                    IF (((( NOT ChargeMode) OR DriveMode) OR SDError_BB) OR (BoxAvailable = 0.0)) AND ( NOT HV_REL_ON_BB) THEN 
                        (* Transition: '<S53>:21' *)
                        (* Exit Internal 'CHARGE': '<S53>:46' *)
                        is_CHARGE := ChiefMaster_IN_NO_ACTIVE_CHILD_jz;
                        is_c66_ChiefMaster := ChiefMaster_IN_Default_d;
                        (* Entry 'Default': '<S53>:9' *)
                        (* '<S53>:9:2' REQ_IMD_ON = false; *)
                        REQ_IMD_ON := FALSE;
                        (* '<S53>:9:3' IMD_State = uint8(0); *)
                        IMD_State := 0;
                    ELSE 

                        CASE is_CHARGE OF
                            ChiefMaster_IN_CHARGE_c: 
                                (* During 'CHARGE': '<S53>:13' *)
                                (* '<S53>:32:1' sf_internal_predicateOutput = InsulationReadyOK == true &&... *)
                                (* '<S53>:32:2' MinVtgBB == BattNo &&... *)
                                (* '<S53>:32:3' HV_ON_BB == false; *)

                                IF (InsulationReadyOK AND (MinVtgBB = BattNo)) AND ( NOT HV_ON_BB) THEN 
                                    (* Transition: '<S53>:32' *)
                                    is_CHARGE := ChiefMaster_IN_IMD_ON_b;
                                    (* Entry 'IMD_ON': '<S53>:31' *)
                                    (* '<S53>:31:2' REQ_IMD_ON = true; *)
                                    REQ_IMD_ON := TRUE;
                                    (* '<S53>:31:3' IMD_State = uint8(5); *)
                                    IMD_State := 5;
                                ELSE 
                                    (* '<S53>:34:1' sf_internal_predicateOutput = (InsulationReadyOK == true && MinVtgBB ~=  BattNo) ||... *)
                                    (* '<S53>:34:2'  HV_ON_BB == true; *)

                                    IF (InsulationReadyOK AND (MinVtgBB <> BattNo)) OR HV_ON_BB THEN 
                                        (* Transition: '<S53>:34' *)
                                        is_CHARGE := ChiefMaster_IN_IMD_OFF_m;
                                        (* Entry 'IMD_OFF': '<S53>:33' *)
                                        (* '<S53>:33:2' REQ_IMD_ON = false; *)
                                        REQ_IMD_ON := FALSE;
                                        (* '<S53>:33:3' IMD_State = uint8(6); *)
                                        IMD_State := 6;
                                    ELSE 
                                        (* '<S53>:13:2' REQ_IMD_ON = true; *)
                                        REQ_IMD_ON := TRUE;
                                        (* '<S53>:13:3' IMD_State = uint8(4); *)
                                        IMD_State := 4;
                                    END_IF;

                                END_IF;

                            ChiefMaster_IN_IMD_OFF_m: 
                                (* During 'IMD_OFF': '<S53>:33' *)
                                (* '<S53>:75:1' sf_internal_predicateOutput = MinVtgBB == BattNo &&... *)
                                (* '<S53>:75:2' IMD_Active_BB1 == false &&... *)
                                (* '<S53>:75:3' IMD_Active_BB2 == false &&... *)
                                (* '<S53>:75:4' IMD_Active_BB3 == false &&... *)
                                (* '<S53>:75:5' IsolationMeasurementRequest == true; *)

                                IF ((((MinVtgBB = BattNo) AND ( NOT IMD_Active_BB1)) AND ( NOT IMD_Active_BB2)) AND ( NOT IMD_Active_BB3)) AND IsolationMeasurementRequest THEN 
                                    (* Transition: '<S53>:75' *)
                                    is_CHARGE := ChiefMaster_IN_IMD_ON_b;
                                    (* Entry 'IMD_ON': '<S53>:31' *)
                                    (* '<S53>:31:2' REQ_IMD_ON = true; *)
                                    REQ_IMD_ON := TRUE;
                                    (* '<S53>:31:3' IMD_State = uint8(5); *)
                                    IMD_State := 5;
                                ELSE 
                                    (* '<S53>:33:2' REQ_IMD_ON = false; *)
                                    REQ_IMD_ON := FALSE;
                                    (* '<S53>:33:3' IMD_State = uint8(6); *)
                                    IMD_State := 6;
                                END_IF;

                            ELSE
                                (* During 'IMD_ON': '<S53>:31' *)
                                (* '<S53>:87:1' sf_internal_predicateOutput = HV_ON_BB == true &&... *)
                                (* '<S53>:87:2' IsolationMeasurementRequest == false; *)

                                IF HV_ON_BB AND ( NOT IsolationMeasurementRequest) THEN 
                                    (* Transition: '<S53>:87' *)
                                    is_CHARGE := ChiefMaster_IN_IMD_OFF_m;
                                    (* Entry 'IMD_OFF': '<S53>:33' *)
                                    (* '<S53>:33:2' REQ_IMD_ON = false; *)
                                    REQ_IMD_ON := FALSE;
                                    (* '<S53>:33:3' IMD_State = uint8(6); *)
                                    IMD_State := 6;
                                ELSE 
                                    (* '<S53>:31:2' REQ_IMD_ON = true; *)
                                    REQ_IMD_ON := TRUE;
                                    (* '<S53>:31:3' IMD_State = uint8(5); *)
                                    IMD_State := 5;
                                END_IF;

                        END_CASE;

                    END_IF;

                ChiefMaster_IN_DRIVE_k: 
                    (* During 'DRIVE': '<S53>:62' *)
                    (* '<S53>:27:1' sf_internal_predicateOutput = ((DriveMode == false || ChargeMode == true ||... *)
                    (* '<S53>:27:2' SDError_BB == true || BoxAvailable==false) &&... *)
                    (* '<S53>:27:3' HV_REL_ON_BB == false); *)

                    IF (((( NOT DriveMode) OR ChargeMode) OR SDError_BB) OR (BoxAvailable = 0.0)) AND ( NOT HV_REL_ON_BB) THEN 
                        (* Transition: '<S53>:27' *)
                        (* Exit Internal 'DRIVE': '<S53>:62' *)
                        is_DRIVE := ChiefMaster_IN_NO_ACTIVE_CHILD_jz;
                        is_c66_ChiefMaster := ChiefMaster_IN_Default_d;
                        (* Entry 'Default': '<S53>:9' *)
                        (* '<S53>:9:2' REQ_IMD_ON = false; *)
                        REQ_IMD_ON := FALSE;
                        (* '<S53>:9:3' IMD_State = uint8(0); *)
                        IMD_State := 0;
                    ELSE 

                        CASE is_DRIVE OF
                            ChiefMaster_IN_DRIVE_ke: 
                                (* During 'DRIVE': '<S53>:63' *)
                                (* '<S53>:67:1' sf_internal_predicateOutput = InsulationReadyOK == true &&... *)
                                (* '<S53>:67:2' MaxVtgBB == BattNo &&... *)
                                (* '<S53>:67:3' HV_ON_BB == false; *)

                                IF (InsulationReadyOK AND (MaxVtgBB = BattNo)) AND ( NOT HV_ON_BB) THEN 
                                    (* Transition: '<S53>:67' *)
                                    is_DRIVE := ChiefMaster_IN_IMD_ON_b;
                                    (* Entry 'IMD_ON': '<S53>:64' *)
                                    (* '<S53>:64:2' REQ_IMD_ON = true; *)
                                    REQ_IMD_ON := TRUE;
                                    (* '<S53>:64:3' IMD_State = uint8(2); *)
                                    IMD_State := 2;
                                ELSE 
                                    (* '<S53>:68:1' sf_internal_predicateOutput = (InsulationReadyOK == true && MaxVtgBB ~=  BattNo)  ||... *)
                                    (* '<S53>:68:2' HV_ON_BB == true; *)

                                    IF (InsulationReadyOK AND (MaxVtgBB <> BattNo)) OR HV_ON_BB THEN 
                                        (* Transition: '<S53>:68' *)
                                        is_DRIVE := ChiefMaster_IN_IMD_OFF_m;
                                        (* Entry 'IMD_OFF': '<S53>:65' *)
                                        (* '<S53>:65:2' REQ_IMD_ON = false; *)
                                        REQ_IMD_ON := FALSE;
                                        (* '<S53>:65:3' IMD_State = uint8(3); *)
                                        IMD_State := 3;
                                    ELSE 
                                        (* '<S53>:63:2' REQ_IMD_ON = true; *)
                                        REQ_IMD_ON := TRUE;
                                        (* '<S53>:63:3' IMD_State = uint8(1); *)
                                        IMD_State := 1;
                                    END_IF;

                                END_IF;

                            ChiefMaster_IN_IMD_OFF_m: 
                                (* During 'IMD_OFF': '<S53>:65' *)
                                (* '<S53>:77:1' sf_internal_predicateOutput = MaxVtgBB == BattNo &&... *)
                                (* '<S53>:77:2' IMD_Active_BB1 == false &&... *)
                                (* '<S53>:77:3' IMD_Active_BB2 == false &&... *)
                                (* '<S53>:77:4' IMD_Active_BB3 == false &&... *)
                                (* '<S53>:77:5' IsolationMeasurementRequest == true; *)

                                IF ((((MaxVtgBB = BattNo) AND ( NOT IMD_Active_BB1)) AND ( NOT IMD_Active_BB2)) AND ( NOT IMD_Active_BB3)) AND IsolationMeasurementRequest THEN 
                                    (* Transition: '<S53>:77' *)
                                    is_DRIVE := ChiefMaster_IN_IMD_ON_b;
                                    (* Entry 'IMD_ON': '<S53>:64' *)
                                    (* '<S53>:64:2' REQ_IMD_ON = true; *)
                                    REQ_IMD_ON := TRUE;
                                    (* '<S53>:64:3' IMD_State = uint8(2); *)
                                    IMD_State := 2;
                                ELSE 
                                    (* '<S53>:65:2' REQ_IMD_ON = false; *)
                                    REQ_IMD_ON := FALSE;
                                    (* '<S53>:65:3' IMD_State = uint8(3); *)
                                    IMD_State := 3;
                                END_IF;

                            ELSE
                                (* During 'IMD_ON': '<S53>:64' *)
                                (* '<S53>:88:1' sf_internal_predicateOutput = HV_ON_BB == true &&... *)
                                (* '<S53>:88:2' IsolationMeasurementRequest == false; *)

                                IF HV_ON_BB AND ( NOT IsolationMeasurementRequest) THEN 
                                    (* Transition: '<S53>:88' *)
                                    is_DRIVE := ChiefMaster_IN_IMD_OFF_m;
                                    (* Entry 'IMD_OFF': '<S53>:65' *)
                                    (* '<S53>:65:2' REQ_IMD_ON = false; *)
                                    REQ_IMD_ON := FALSE;
                                    (* '<S53>:65:3' IMD_State = uint8(3); *)
                                    IMD_State := 3;
                                ELSE 
                                    (* '<S53>:64:2' REQ_IMD_ON = true; *)
                                    REQ_IMD_ON := TRUE;
                                    (* '<S53>:64:3' IMD_State = uint8(2); *)
                                    IMD_State := 2;
                                END_IF;

                        END_CASE;

                    END_IF;

                ELSE
                    (* During 'Default': '<S53>:9' *)
                    (* '<S53>:14:1' sf_internal_predicateOutput = ChargeMode == true && DriveMode == false &&... *)
                    (* '<S53>:14:2'  SDError_BB == false && BoxAvailable==true; *)
                    tmp :=  NOT SDError_BB;

                    IF ((ChargeMode AND ( NOT DriveMode)) AND tmp) AND (BoxAvailable = 1.0) THEN 
                        (* Transition: '<S53>:14' *)
                        is_c66_ChiefMaster := ChiefMaster_IN_CHARGE_c;
                        (* Entry Internal 'CHARGE': '<S53>:46' *)
                        (* Transition: '<S53>:47' *)
                        is_CHARGE := ChiefMaster_IN_CHARGE_c;
                        (* Entry 'CHARGE': '<S53>:13' *)
                        (* '<S53>:13:2' REQ_IMD_ON = true; *)
                        REQ_IMD_ON := TRUE;
                        (* '<S53>:13:3' IMD_State = uint8(4); *)
                        IMD_State := 4;
                    ELSE 
                        (* '<S53>:18:1' sf_internal_predicateOutput = DriveMode == true && ChargeMode == false &&... *)
                        (* '<S53>:18:2'  SDError_BB == false && BoxAvailable==true; *)

                        IF ((DriveMode AND ( NOT ChargeMode)) AND tmp) AND (BoxAvailable = 1.0) THEN 
                            (* Transition: '<S53>:18' *)
                            is_c66_ChiefMaster := ChiefMaster_IN_DRIVE_k;
                            (* Entry Internal 'DRIVE': '<S53>:62' *)
                            (* Transition: '<S53>:66' *)
                            is_DRIVE := ChiefMaster_IN_DRIVE_ke;
                            (* Entry 'DRIVE': '<S53>:63' *)
                            (* '<S53>:63:2' REQ_IMD_ON = true; *)
                            REQ_IMD_ON := TRUE;
                            (* '<S53>:63:3' IMD_State = uint8(1); *)
                            IMD_State := 1;
                        ELSE 
                            (* '<S53>:9:2' REQ_IMD_ON = false; *)
                            REQ_IMD_ON := FALSE;
                            (* '<S53>:9:3' IMD_State = uint8(0); *)
                            IMD_State := 0;
                        END_IF;

                    END_IF;

            END_CASE;

        END_IF;

        (* End of Chart: '<S48>/Chart_REQ_IMD_ON_BB2' *)
END_CASE;

END_FUNCTION_BLOCK

// Device/Application/Chart_REQ_IMD_ON_BB3
FUNCTION_BLOCK Chart_REQ_IMD_ON_BB3
VAR_INPUT
	ssMethodType: SINT;
	ChargeMode: BOOL;
	DriveMode: BOOL;
	InsulationReadyOK: BOOL;
	MaxVtgBB: REAL;
	MinVtgBB: REAL;
	SDError_BB: BOOL;
	BattNo: REAL;
	HV_ON_BB: BOOL;
	IMD_Active_BB2: BOOL;
	IMD_Active_BB3: BOOL;
	IMD_Active_BB1: BOOL;
	HV_REL_ON_BB: BOOL;
	BoxAvailable: LREAL;
	IsolationMeasurementRequest: BOOL;
END_VAR
VAR_OUTPUT
	REQ_IMD_ON: BOOL;
	IMD_State: USINT;
END_VAR
VAR
	is_c67_ChiefMaster: USINT;
	is_active_c67_ChiefMaster: USINT;
	is_DRIVE: USINT;
	is_CHARGE: USINT;
	tmp: BOOL;
END_VAR



CASE ssMethodType OF
    SS_INITIALIZE: 
        is_CHARGE := ChiefMaster_IN_NO_ACTIVE_CHILD_g;
        is_DRIVE := ChiefMaster_IN_NO_ACTIVE_CHILD_g;
        is_active_c67_ChiefMaster := 0;
        is_c67_ChiefMaster := ChiefMaster_IN_NO_ACTIVE_CHILD_g;
        REQ_IMD_ON := FALSE;
        IMD_State := 0;
    SS_OUTPUT: 
        (* Chart: '<S48>/Chart_REQ_IMD_ON_BB3' *)
        (* Gateway: ChiefMaster/Flow Logic/IMD Control/InsulationMonitoringReq/Chart_REQ_IMD_ON_BB3 *)
        (* During: ChiefMaster/Flow Logic/IMD Control/InsulationMonitoringReq/Chart_REQ_IMD_ON_BB3 *)

        IF is_active_c67_ChiefMaster = 0 THEN 
            (* Entry: ChiefMaster/Flow Logic/IMD Control/InsulationMonitoringReq/Chart_REQ_IMD_ON_BB3 *)
            is_active_c67_ChiefMaster := 1;
            (* Entry Internal: ChiefMaster/Flow Logic/IMD Control/InsulationMonitoringReq/Chart_REQ_IMD_ON_BB3 *)
            (* Transition: '<S54>:10' *)
            is_c67_ChiefMaster := ChiefMaster_IN_Default_j;
            (* Entry 'Default': '<S54>:9' *)
            (* '<S54>:9:2' REQ_IMD_ON = false; *)
            REQ_IMD_ON := FALSE;
            (* '<S54>:9:3' IMD_State = uint8(0); *)
            IMD_State := 0;
        ELSE 

            CASE is_c67_ChiefMaster OF
                ChiefMaster_IN_CHARGE_a: 
                    (* During 'CHARGE': '<S54>:46' *)
                    (* '<S54>:21:1' sf_internal_predicateOutput = ((ChargeMode == false || DriveMode == true ||... *)
                    (* '<S54>:21:2'  SDError_BB == true || BoxAvailable==false) &&... *)
                    (* '<S54>:21:3' HV_REL_ON_BB == false); *)

                    IF (((( NOT ChargeMode) OR DriveMode) OR SDError_BB) OR (BoxAvailable = 0.0)) AND ( NOT HV_REL_ON_BB) THEN 
                        (* Transition: '<S54>:21' *)
                        (* Exit Internal 'CHARGE': '<S54>:46' *)
                        is_CHARGE := ChiefMaster_IN_NO_ACTIVE_CHILD_g;
                        is_c67_ChiefMaster := ChiefMaster_IN_Default_j;
                        (* Entry 'Default': '<S54>:9' *)
                        (* '<S54>:9:2' REQ_IMD_ON = false; *)
                        REQ_IMD_ON := FALSE;
                        (* '<S54>:9:3' IMD_State = uint8(0); *)
                        IMD_State := 0;
                    ELSE 

                        CASE is_CHARGE OF
                            ChiefMaster_IN_CHARGE_a: 
                                (* During 'CHARGE': '<S54>:13' *)
                                (* '<S54>:32:1' sf_internal_predicateOutput = InsulationReadyOK == true &&... *)
                                (* '<S54>:32:2' MinVtgBB == BattNo &&... *)
                                (* '<S54>:32:3' HV_ON_BB == false; *)

                                IF (InsulationReadyOK AND (MinVtgBB = BattNo)) AND ( NOT HV_ON_BB) THEN 
                                    (* Transition: '<S54>:32' *)
                                    is_CHARGE := ChiefMaster_IN_IMD_ON_k;
                                    (* Entry 'IMD_ON': '<S54>:31' *)
                                    (* '<S54>:31:2' REQ_IMD_ON = true; *)
                                    REQ_IMD_ON := TRUE;
                                    (* '<S54>:31:3' IMD_State = uint8(5); *)
                                    IMD_State := 5;
                                ELSE 
                                    (* '<S54>:34:1' sf_internal_predicateOutput = (InsulationReadyOK == true && MinVtgBB ~=  BattNo) ||... *)
                                    (* '<S54>:34:2'  HV_ON_BB == true; *)

                                    IF (InsulationReadyOK AND (MinVtgBB <> BattNo)) OR HV_ON_BB THEN 
                                        (* Transition: '<S54>:34' *)
                                        is_CHARGE := ChiefMaster_IN_IMD_OFF_a;
                                        (* Entry 'IMD_OFF': '<S54>:33' *)
                                        (* '<S54>:33:2' REQ_IMD_ON = false; *)
                                        REQ_IMD_ON := FALSE;
                                        (* '<S54>:33:3' IMD_State = uint8(6); *)
                                        IMD_State := 6;
                                    ELSE 
                                        (* '<S54>:13:2' REQ_IMD_ON = true; *)
                                        REQ_IMD_ON := TRUE;
                                        (* '<S54>:13:3' IMD_State = uint8(4); *)
                                        IMD_State := 4;
                                    END_IF;

                                END_IF;

                            ChiefMaster_IN_IMD_OFF_a: 
                                (* During 'IMD_OFF': '<S54>:33' *)
                                (* '<S54>:75:1' sf_internal_predicateOutput = MinVtgBB == BattNo &&... *)
                                (* '<S54>:75:2' IMD_Active_BB1 == false &&... *)
                                (* '<S54>:75:3' IMD_Active_BB2 == false &&... *)
                                (* '<S54>:75:4' IMD_Active_BB3 == false &&... *)
                                (* '<S54>:75:5' IsolationMeasurementRequest == true; *)

                                IF ((((MinVtgBB = BattNo) AND ( NOT IMD_Active_BB1)) AND ( NOT IMD_Active_BB2)) AND ( NOT IMD_Active_BB3)) AND IsolationMeasurementRequest THEN 
                                    (* Transition: '<S54>:75' *)
                                    is_CHARGE := ChiefMaster_IN_IMD_ON_k;
                                    (* Entry 'IMD_ON': '<S54>:31' *)
                                    (* '<S54>:31:2' REQ_IMD_ON = true; *)
                                    REQ_IMD_ON := TRUE;
                                    (* '<S54>:31:3' IMD_State = uint8(5); *)
                                    IMD_State := 5;
                                ELSE 
                                    (* '<S54>:33:2' REQ_IMD_ON = false; *)
                                    REQ_IMD_ON := FALSE;
                                    (* '<S54>:33:3' IMD_State = uint8(6); *)
                                    IMD_State := 6;
                                END_IF;

                            ELSE
                                (* During 'IMD_ON': '<S54>:31' *)
                                (* '<S54>:87:1' sf_internal_predicateOutput = HV_ON_BB == true &&... *)
                                (* '<S54>:87:2' IsolationMeasurementRequest == false; *)

                                IF HV_ON_BB AND ( NOT IsolationMeasurementRequest) THEN 
                                    (* Transition: '<S54>:87' *)
                                    is_CHARGE := ChiefMaster_IN_IMD_OFF_a;
                                    (* Entry 'IMD_OFF': '<S54>:33' *)
                                    (* '<S54>:33:2' REQ_IMD_ON = false; *)
                                    REQ_IMD_ON := FALSE;
                                    (* '<S54>:33:3' IMD_State = uint8(6); *)
                                    IMD_State := 6;
                                ELSE 
                                    (* '<S54>:31:2' REQ_IMD_ON = true; *)
                                    REQ_IMD_ON := TRUE;
                                    (* '<S54>:31:3' IMD_State = uint8(5); *)
                                    IMD_State := 5;
                                END_IF;

                        END_CASE;

                    END_IF;

                ChiefMaster_IN_DRIVE_e: 
                    (* During 'DRIVE': '<S54>:62' *)
                    (* '<S54>:27:1' sf_internal_predicateOutput = ((DriveMode == false || ChargeMode == true ||... *)
                    (* '<S54>:27:2' SDError_BB == true || BoxAvailable==false) &&... *)
                    (* '<S54>:27:3' HV_REL_ON_BB == false); *)

                    IF (((( NOT DriveMode) OR ChargeMode) OR SDError_BB) OR (BoxAvailable = 0.0)) AND ( NOT HV_REL_ON_BB) THEN 
                        (* Transition: '<S54>:27' *)
                        (* Exit Internal 'DRIVE': '<S54>:62' *)
                        is_DRIVE := ChiefMaster_IN_NO_ACTIVE_CHILD_g;
                        is_c67_ChiefMaster := ChiefMaster_IN_Default_j;
                        (* Entry 'Default': '<S54>:9' *)
                        (* '<S54>:9:2' REQ_IMD_ON = false; *)
                        REQ_IMD_ON := FALSE;
                        (* '<S54>:9:3' IMD_State = uint8(0); *)
                        IMD_State := 0;
                    ELSE 

                        CASE is_DRIVE OF
                            ChiefMaster_IN_DRIVE_e3: 
                                (* During 'DRIVE': '<S54>:63' *)
                                (* '<S54>:67:1' sf_internal_predicateOutput = InsulationReadyOK == true &&... *)
                                (* '<S54>:67:2' MaxVtgBB == BattNo &&... *)
                                (* '<S54>:67:3' HV_ON_BB == false; *)

                                IF (InsulationReadyOK AND (MaxVtgBB = BattNo)) AND ( NOT HV_ON_BB) THEN 
                                    (* Transition: '<S54>:67' *)
                                    is_DRIVE := ChiefMaster_IN_IMD_ON_k;
                                    (* Entry 'IMD_ON': '<S54>:64' *)
                                    (* '<S54>:64:2' REQ_IMD_ON = true; *)
                                    REQ_IMD_ON := TRUE;
                                    (* '<S54>:64:3' IMD_State = uint8(2); *)
                                    IMD_State := 2;
                                ELSE 
                                    (* '<S54>:68:1' sf_internal_predicateOutput = (InsulationReadyOK == true && MaxVtgBB ~=  BattNo)  ||... *)
                                    (* '<S54>:68:2' HV_ON_BB == true; *)

                                    IF (InsulationReadyOK AND (MaxVtgBB <> BattNo)) OR HV_ON_BB THEN 
                                        (* Transition: '<S54>:68' *)
                                        is_DRIVE := ChiefMaster_IN_IMD_OFF_a;
                                        (* Entry 'IMD_OFF': '<S54>:65' *)
                                        (* '<S54>:65:2' REQ_IMD_ON = false; *)
                                        REQ_IMD_ON := FALSE;
                                        (* '<S54>:65:3' IMD_State = uint8(3); *)
                                        IMD_State := 3;
                                    ELSE 
                                        (* '<S54>:63:2' REQ_IMD_ON = true; *)
                                        REQ_IMD_ON := TRUE;
                                        (* '<S54>:63:3' IMD_State = uint8(1); *)
                                        IMD_State := 1;
                                    END_IF;

                                END_IF;

                            ChiefMaster_IN_IMD_OFF_a: 
                                (* During 'IMD_OFF': '<S54>:65' *)
                                (* '<S54>:77:1' sf_internal_predicateOutput = MaxVtgBB == BattNo &&... *)
                                (* '<S54>:77:2' IMD_Active_BB1 == false &&... *)
                                (* '<S54>:77:3' IMD_Active_BB2 == false &&... *)
                                (* '<S54>:77:4' IMD_Active_BB3 == false &&... *)
                                (* '<S54>:77:5' IsolationMeasurementRequest == true; *)

                                IF ((((MaxVtgBB = BattNo) AND ( NOT IMD_Active_BB1)) AND ( NOT IMD_Active_BB2)) AND ( NOT IMD_Active_BB3)) AND IsolationMeasurementRequest THEN 
                                    (* Transition: '<S54>:77' *)
                                    is_DRIVE := ChiefMaster_IN_IMD_ON_k;
                                    (* Entry 'IMD_ON': '<S54>:64' *)
                                    (* '<S54>:64:2' REQ_IMD_ON = true; *)
                                    REQ_IMD_ON := TRUE;
                                    (* '<S54>:64:3' IMD_State = uint8(2); *)
                                    IMD_State := 2;
                                ELSE 
                                    (* '<S54>:65:2' REQ_IMD_ON = false; *)
                                    REQ_IMD_ON := FALSE;
                                    (* '<S54>:65:3' IMD_State = uint8(3); *)
                                    IMD_State := 3;
                                END_IF;

                            ELSE
                                (* During 'IMD_ON': '<S54>:64' *)
                                (* '<S54>:88:1' sf_internal_predicateOutput = HV_ON_BB == true &&... *)
                                (* '<S54>:88:2' IsolationMeasurementRequest == false; *)

                                IF HV_ON_BB AND ( NOT IsolationMeasurementRequest) THEN 
                                    (* Transition: '<S54>:88' *)
                                    is_DRIVE := ChiefMaster_IN_IMD_OFF_a;
                                    (* Entry 'IMD_OFF': '<S54>:65' *)
                                    (* '<S54>:65:2' REQ_IMD_ON = false; *)
                                    REQ_IMD_ON := FALSE;
                                    (* '<S54>:65:3' IMD_State = uint8(3); *)
                                    IMD_State := 3;
                                ELSE 
                                    (* '<S54>:64:2' REQ_IMD_ON = true; *)
                                    REQ_IMD_ON := TRUE;
                                    (* '<S54>:64:3' IMD_State = uint8(2); *)
                                    IMD_State := 2;
                                END_IF;

                        END_CASE;

                    END_IF;

                ELSE
                    (* During 'Default': '<S54>:9' *)
                    (* '<S54>:14:1' sf_internal_predicateOutput = ChargeMode == true && DriveMode == false &&... *)
                    (* '<S54>:14:2'  SDError_BB == false && BoxAvailable==true; *)
                    tmp :=  NOT SDError_BB;

                    IF ((ChargeMode AND ( NOT DriveMode)) AND tmp) AND (BoxAvailable = 1.0) THEN 
                        (* Transition: '<S54>:14' *)
                        is_c67_ChiefMaster := ChiefMaster_IN_CHARGE_a;
                        (* Entry Internal 'CHARGE': '<S54>:46' *)
                        (* Transition: '<S54>:47' *)
                        is_CHARGE := ChiefMaster_IN_CHARGE_a;
                        (* Entry 'CHARGE': '<S54>:13' *)
                        (* '<S54>:13:2' REQ_IMD_ON = true; *)
                        REQ_IMD_ON := TRUE;
                        (* '<S54>:13:3' IMD_State = uint8(4); *)
                        IMD_State := 4;
                    ELSE 
                        (* '<S54>:18:1' sf_internal_predicateOutput = DriveMode == true && ChargeMode == false &&... *)
                        (* '<S54>:18:2'  SDError_BB == false && BoxAvailable==true; *)

                        IF ((DriveMode AND ( NOT ChargeMode)) AND tmp) AND (BoxAvailable = 1.0) THEN 
                            (* Transition: '<S54>:18' *)
                            is_c67_ChiefMaster := ChiefMaster_IN_DRIVE_e;
                            (* Entry Internal 'DRIVE': '<S54>:62' *)
                            (* Transition: '<S54>:66' *)
                            is_DRIVE := ChiefMaster_IN_DRIVE_e3;
                            (* Entry 'DRIVE': '<S54>:63' *)
                            (* '<S54>:63:2' REQ_IMD_ON = true; *)
                            REQ_IMD_ON := TRUE;
                            (* '<S54>:63:3' IMD_State = uint8(1); *)
                            IMD_State := 1;
                        ELSE 
                            (* '<S54>:9:2' REQ_IMD_ON = false; *)
                            REQ_IMD_ON := FALSE;
                            (* '<S54>:9:3' IMD_State = uint8(0); *)
                            IMD_State := 0;
                        END_IF;

                    END_IF;

            END_CASE;

        END_IF;

        (* End of Chart: '<S48>/Chart_REQ_IMD_ON_BB3' *)
END_CASE;

END_FUNCTION_BLOCK

// Device/Application/PLC_CODER_TIMER
FUNCTION_BLOCK PLC_CODER_TIMER
VAR_INPUT
	timerAction: INT;
	maxTime: DINT;
END_VAR
VAR_OUTPUT
	done: BOOL;
END_VAR
VAR
	plcTimer: TON;
	plcTimerExpired: BOOL;
END_VAR


CASE timerAction OF
    1:
        (* RESET *)
        plcTimer(IN:=FALSE, PT:=T#0ms);
        plcTimerExpired := FALSE;
        done := FALSE;
    2:
        (* AFTER *)
        IF (NOT(plcTimerExpired)) THEN
            plcTimer(IN:=TRUE, PT:=DINT_TO_TIME(maxTime));
        END_IF;
        plcTimerExpired := plcTimer.Q;
        done := plcTimerExpired;
    3:
        (* BEFORE *)
        IF (NOT(plcTimerExpired)) THEN
            plcTimer(IN:=TRUE, PT:=DINT_TO_TIME(maxTime));
        END_IF;
        plcTimerExpired := plcTimer.Q;
        done := NOT(plcTimerExpired);
END_CASE;

END_FUNCTION_BLOCK

// Device/Application/PLC_BOOL_TO_LREAL
FUNCTION PLC_BOOL_TO_LREAL : LREAL
VAR_INPUT
	in: BOOL;
END_VAR
VAR
END_VAR



IF in THEN 
    PLC_BOOL_TO_LREAL := 1.0;
ELSE 
    PLC_BOOL_TO_LREAL := 0.0;
END_IF;

END_FUNCTION

// Device/Application/rt_floord
FUNCTION rt_floord : LREAL
VAR_INPUT
	u: LREAL;
END_VAR
VAR
END_VAR


rt_floord := DINT_TO_LREAL(TRUNC(u));

IF u = rt_floord THEN 
    rt_floord := u;
ELSIF u < 0.0 THEN 
    rt_floord := rt_floord - 1.0;
END_IF;

END_FUNCTION

// Device/Application/rt_floorf
FUNCTION rt_floorf : REAL
VAR_INPUT
	u: REAL;
END_VAR
VAR
END_VAR


rt_floorf := DINT_TO_REAL(TRUNC(u));

IF u = rt_floorf THEN 
    rt_floorf := u;
ELSIF u < 0.0 THEN 
    rt_floorf := rt_floorf - 1.0;
END_IF;

END_FUNCTION

// Device/Application/Chart_m
FUNCTION_BLOCK Chart_m
VAR_INPUT
	ssMethodType: SINT;
	In: BOOL;
	KL15_CM_Reset: BOOL;
END_VAR
VAR_OUTPUT
	Out: BOOL;
END_VAR
VAR
	temporalCounter_i1: PLC_CODER_TIMER;
	is_c45_ChiefMaster: USINT;
	is_active_c45_ChiefMaster: USINT;
END_VAR



CASE ssMethodType OF
    SS_INITIALIZE: 
        temporalCounter_i1(timerAction := 1, maxTime := 0);
        is_active_c45_ChiefMaster := 0;
        is_c45_ChiefMaster := ChiefMaster_IN_NO_ACTIVE_CHILD_mp;
        Out := FALSE;
    SS_OUTPUT: 
        (* Chart: '<S56>/Chart' *)
        (* Gateway: ChiefMaster/Flow Logic/KL15/System_KL15/Subsystem/Chart *)
        (* During: ChiefMaster/Flow Logic/KL15/System_KL15/Subsystem/Chart *)

        IF is_active_c45_ChiefMaster = 0 THEN 
            (* Entry: ChiefMaster/Flow Logic/KL15/System_KL15/Subsystem/Chart *)
            is_active_c45_ChiefMaster := 1;
            (* Entry Internal: ChiefMaster/Flow Logic/KL15/System_KL15/Subsystem/Chart *)
            (* Transition: '<S59>:2' *)
            is_c45_ChiefMaster := ChiefMaster_IN_Default_o;
            temporalCounter_i1(timerAction := 1, maxTime := 0);
            (* Entry 'Default': '<S59>:1' *)
            (* '<S59>:1:2' Out = false *)
            Out := FALSE;
        ELSE 

            CASE is_c45_ChiefMaster OF
                ChiefMaster_IN_Default_o: 
                    (* During 'Default': '<S59>:1' *)
                    (* '<S59>:4:1' sf_internal_predicateOutput = KL15_CM_Reset == false &&... *)
                    (* '<S59>:4:2' after(100,msec); *)

                    IF  NOT KL15_CM_Reset THEN 
                        temporalCounter_i1(timerAction := 2, maxTime := 100);

                        IF temporalCounter_i1.done THEN 
                            (* Transition: '<S59>:4' *)
                            is_c45_ChiefMaster := ChiefMaster_IN_hold_g;
                            (* Entry 'hold': '<S59>:7' *)
                            (* '<S59>:7:2' Out = In *)
                            Out := In;
                        ELSE 
                            (* '<S59>:1:2' Out = false *)
                            Out := FALSE;
                        END_IF;

                    ELSE 
                        (* '<S59>:1:2' Out = false *)
                        Out := FALSE;
                    END_IF;

                ELSE
                    (* During 'hold': '<S59>:7' *)
                    (* '<S59>:7:2' Out = In *)
                    Out := In;
            END_CASE;

        END_IF;

        (* End of Chart: '<S56>/Chart' *)
END_CASE;

END_FUNCTION_BLOCK

// Device/Application/ChartBatt1
FUNCTION_BLOCK ChartBatt1
VAR_INPUT
	ssMethodType: SINT;
	BattAvailable_LiBa: BOOL;
	BattAvailable_Actia: BOOL;
END_VAR
VAR_OUTPUT
	BattSelect: LREAL;
END_VAR
VAR
	is_c9_ChiefMaster: USINT;
	is_active_c9_ChiefMaster: USINT;
END_VAR



CASE ssMethodType OF
    SS_INITIALIZE: 
        is_active_c9_ChiefMaster := 0;
        is_c9_ChiefMaster := ChiefMaster_IN_NO_ACTIVE_CHILD_i3;
        BattSelect := 0.0;
    SS_OUTPUT: 
        (* Chart: '<S675>/ChartBatt1' *)
        (* Gateway: ChiefMaster/Input Translation/Battery Selection/ChartBatt1 *)
        (* During: ChiefMaster/Input Translation/Battery Selection/ChartBatt1 *)

        IF is_active_c9_ChiefMaster = 0 THEN 
            (* Entry: ChiefMaster/Input Translation/Battery Selection/ChartBatt1 *)
            is_active_c9_ChiefMaster := 1;
            (* Entry Internal: ChiefMaster/Input Translation/Battery Selection/ChartBatt1 *)
            (* Transition: '<S679>:2' *)
            is_c9_ChiefMaster := ChiefMaster_IN_Default_at;
            (* Entry 'Default': '<S679>:1' *)
            (* '<S679>:1:2' BattSelect=0; *)
            BattSelect := 0.0;
        ELSE 

            CASE is_c9_ChiefMaster OF
                ChiefMaster_IN_Actia: 
                    (* During 'Actia': '<S679>:3' *)
                    (* '<S679>:7:1' sf_internal_predicateOutput = BattAvailable_Actia == false; *)

                    IF  NOT BattAvailable_Actia THEN 
                        (* Transition: '<S679>:7' *)
                        is_c9_ChiefMaster := ChiefMaster_IN_Default_at;
                        (* Entry 'Default': '<S679>:1' *)
                        (* '<S679>:1:2' BattSelect=0; *)
                        BattSelect := 0.0;
                    ELSE 
                        (* '<S679>:3:2' BattSelect=1; *)
                        BattSelect := 1.0;
                    END_IF;

                ChiefMaster_IN_Default_at: 
                    (* During 'Default': '<S679>:1' *)
                    (* '<S679>:6:1' sf_internal_predicateOutput = BattAvailable_Actia == true &&... *)
                    (* '<S679>:6:2' BattAvailable_LiBa == false; *)

                    IF BattAvailable_Actia AND ( NOT BattAvailable_LiBa) THEN 
                        (* Transition: '<S679>:6' *)
                        is_c9_ChiefMaster := ChiefMaster_IN_Actia;
                        (* Entry 'Actia': '<S679>:3' *)
                        (* '<S679>:3:2' BattSelect=1; *)
                        BattSelect := 1.0;
                    ELSE 
                        (* '<S679>:5:1' sf_internal_predicateOutput = BattAvailable_Actia == false &&... *)
                        (* '<S679>:5:2' BattAvailable_LiBa == true; *)

                        IF ( NOT BattAvailable_Actia) AND BattAvailable_LiBa THEN 
                            (* Transition: '<S679>:5' *)
                            is_c9_ChiefMaster := ChiefMaster_IN_LiBa;
                            (* Entry 'LiBa': '<S679>:4' *)
                            (* '<S679>:4:2' BattSelect = 2; *)
                            BattSelect := 2.0;
                        ELSE 
                            (* '<S679>:1:2' BattSelect=0; *)
                            BattSelect := 0.0;
                        END_IF;

                    END_IF;

                ELSE
                    (* During 'LiBa': '<S679>:4' *)
                    (* '<S679>:8:1' sf_internal_predicateOutput = BattAvailable_LiBa == false; *)

                    IF  NOT BattAvailable_LiBa THEN 
                        (* Transition: '<S679>:8' *)
                        is_c9_ChiefMaster := ChiefMaster_IN_Default_at;
                        (* Entry 'Default': '<S679>:1' *)
                        (* '<S679>:1:2' BattSelect=0; *)
                        BattSelect := 0.0;
                    ELSE 
                        (* '<S679>:4:2' BattSelect = 2; *)
                        BattSelect := 2.0;
                    END_IF;

            END_CASE;

        END_IF;

        (* End of Chart: '<S675>/ChartBatt1' *)
END_CASE;

END_FUNCTION_BLOCK

// Device/Application/Chartbatt2
FUNCTION_BLOCK Chartbatt2
VAR_INPUT
	ssMethodType: SINT;
	BattAvailable_LiBa: BOOL;
	BattAvailable_Actia: BOOL;
END_VAR
VAR_OUTPUT
	BattSelect: LREAL;
END_VAR
VAR
	is_c22_ChiefMaster: USINT;
	is_active_c22_ChiefMaster: USINT;
END_VAR



CASE ssMethodType OF
    SS_INITIALIZE: 
        is_active_c22_ChiefMaster := 0;
        is_c22_ChiefMaster := ChiefMaster_IN_NO_ACTIVE_CHILD_gp;
        BattSelect := 0.0;
    SS_OUTPUT: 
        (* Chart: '<S675>/Chartbatt2' *)
        (* Gateway: ChiefMaster/Input Translation/Battery Selection/Chartbatt2 *)
        (* During: ChiefMaster/Input Translation/Battery Selection/Chartbatt2 *)

        IF is_active_c22_ChiefMaster = 0 THEN 
            (* Entry: ChiefMaster/Input Translation/Battery Selection/Chartbatt2 *)
            is_active_c22_ChiefMaster := 1;
            (* Entry Internal: ChiefMaster/Input Translation/Battery Selection/Chartbatt2 *)
            (* Transition: '<S681>:2' *)
            is_c22_ChiefMaster := ChiefMaster_IN_Default_bc;
            (* Entry 'Default': '<S681>:1' *)
            (* '<S681>:1:2' BattSelect=0; *)
            BattSelect := 0.0;
        ELSE 

            CASE is_c22_ChiefMaster OF
                ChiefMaster_IN_Actia_p: 
                    (* During 'Actia': '<S681>:3' *)
                    (* '<S681>:7:1' sf_internal_predicateOutput = BattAvailable_Actia == false; *)

                    IF  NOT BattAvailable_Actia THEN 
                        (* Transition: '<S681>:7' *)
                        is_c22_ChiefMaster := ChiefMaster_IN_Default_bc;
                        (* Entry 'Default': '<S681>:1' *)
                        (* '<S681>:1:2' BattSelect=0; *)
                        BattSelect := 0.0;
                    ELSE 
                        (* '<S681>:3:2' BattSelect=1; *)
                        BattSelect := 1.0;
                    END_IF;

                ChiefMaster_IN_Default_bc: 
                    (* During 'Default': '<S681>:1' *)
                    (* '<S681>:6:1' sf_internal_predicateOutput = BattAvailable_Actia == true &&... *)
                    (* '<S681>:6:2' BattAvailable_LiBa == false; *)

                    IF BattAvailable_Actia AND ( NOT BattAvailable_LiBa) THEN 
                        (* Transition: '<S681>:6' *)
                        is_c22_ChiefMaster := ChiefMaster_IN_Actia_p;
                        (* Entry 'Actia': '<S681>:3' *)
                        (* '<S681>:3:2' BattSelect=1; *)
                        BattSelect := 1.0;
                    ELSE 
                        (* '<S681>:5:1' sf_internal_predicateOutput = BattAvailable_Actia == false &&... *)
                        (* '<S681>:5:2' BattAvailable_LiBa == true; *)

                        IF ( NOT BattAvailable_Actia) AND BattAvailable_LiBa THEN 
                            (* Transition: '<S681>:5' *)
                            is_c22_ChiefMaster := ChiefMaster_IN_LiBa_d;
                            (* Entry 'LiBa': '<S681>:4' *)
                            (* '<S681>:4:2' BattSelect = 2; *)
                            BattSelect := 2.0;
                        ELSE 
                            (* '<S681>:1:2' BattSelect=0; *)
                            BattSelect := 0.0;
                        END_IF;

                    END_IF;

                ELSE
                    (* During 'LiBa': '<S681>:4' *)
                    (* '<S681>:8:1' sf_internal_predicateOutput = BattAvailable_LiBa == false; *)

                    IF  NOT BattAvailable_LiBa THEN 
                        (* Transition: '<S681>:8' *)
                        is_c22_ChiefMaster := ChiefMaster_IN_Default_bc;
                        (* Entry 'Default': '<S681>:1' *)
                        (* '<S681>:1:2' BattSelect=0; *)
                        BattSelect := 0.0;
                    ELSE 
                        (* '<S681>:4:2' BattSelect = 2; *)
                        BattSelect := 2.0;
                    END_IF;

            END_CASE;

        END_IF;

        (* End of Chart: '<S675>/Chartbatt2' *)
END_CASE;

END_FUNCTION_BLOCK

// Device/Application/ChartBatt3
FUNCTION_BLOCK ChartBatt3
VAR_INPUT
	ssMethodType: SINT;
	BattAvailable_LiBa: BOOL;
	BattAvailable_Actia: BOOL;
END_VAR
VAR_OUTPUT
	BattSelect: LREAL;
END_VAR
VAR
	is_c23_ChiefMaster: USINT;
	is_active_c23_ChiefMaster: USINT;
END_VAR



CASE ssMethodType OF
    SS_INITIALIZE: 
        is_active_c23_ChiefMaster := 0;
        is_c23_ChiefMaster := ChiefMaster_IN_NO_ACTIVE_CHILD_d4;
        BattSelect := 0.0;
    SS_OUTPUT: 
        (* Chart: '<S675>/ChartBatt3' *)
        (* Gateway: ChiefMaster/Input Translation/Battery Selection/ChartBatt3 *)
        (* During: ChiefMaster/Input Translation/Battery Selection/ChartBatt3 *)

        IF is_active_c23_ChiefMaster = 0 THEN 
            (* Entry: ChiefMaster/Input Translation/Battery Selection/ChartBatt3 *)
            is_active_c23_ChiefMaster := 1;
            (* Entry Internal: ChiefMaster/Input Translation/Battery Selection/ChartBatt3 *)
            (* Transition: '<S680>:2' *)
            is_c23_ChiefMaster := ChiefMaster_IN_Default_jw;
            (* Entry 'Default': '<S680>:1' *)
            (* '<S680>:1:2' BattSelect=0; *)
            BattSelect := 0.0;
        ELSE 

            CASE is_c23_ChiefMaster OF
                ChiefMaster_IN_Actia_m: 
                    (* During 'Actia': '<S680>:3' *)
                    (* '<S680>:7:1' sf_internal_predicateOutput = BattAvailable_Actia == false; *)

                    IF  NOT BattAvailable_Actia THEN 
                        (* Transition: '<S680>:7' *)
                        is_c23_ChiefMaster := ChiefMaster_IN_Default_jw;
                        (* Entry 'Default': '<S680>:1' *)
                        (* '<S680>:1:2' BattSelect=0; *)
                        BattSelect := 0.0;
                    ELSE 
                        (* '<S680>:3:2' BattSelect=1; *)
                        BattSelect := 1.0;
                    END_IF;

                ChiefMaster_IN_Default_jw: 
                    (* During 'Default': '<S680>:1' *)
                    (* '<S680>:6:1' sf_internal_predicateOutput = BattAvailable_Actia == true &&... *)
                    (* '<S680>:6:2' BattAvailable_LiBa == false; *)

                    IF BattAvailable_Actia AND ( NOT BattAvailable_LiBa) THEN 
                        (* Transition: '<S680>:6' *)
                        is_c23_ChiefMaster := ChiefMaster_IN_Actia_m;
                        (* Entry 'Actia': '<S680>:3' *)
                        (* '<S680>:3:2' BattSelect=1; *)
                        BattSelect := 1.0;
                    ELSE 
                        (* '<S680>:5:1' sf_internal_predicateOutput = BattAvailable_Actia == false &&... *)
                        (* '<S680>:5:2' BattAvailable_LiBa == true; *)

                        IF ( NOT BattAvailable_Actia) AND BattAvailable_LiBa THEN 
                            (* Transition: '<S680>:5' *)
                            is_c23_ChiefMaster := ChiefMaster_IN_LiBa_h;
                            (* Entry 'LiBa': '<S680>:4' *)
                            (* '<S680>:4:2' BattSelect = 2; *)
                            BattSelect := 2.0;
                        ELSE 
                            (* '<S680>:1:2' BattSelect=0; *)
                            BattSelect := 0.0;
                        END_IF;

                    END_IF;

                ELSE
                    (* During 'LiBa': '<S680>:4' *)
                    (* '<S680>:8:1' sf_internal_predicateOutput = BattAvailable_LiBa == false; *)

                    IF  NOT BattAvailable_LiBa THEN 
                        (* Transition: '<S680>:8' *)
                        is_c23_ChiefMaster := ChiefMaster_IN_Default_jw;
                        (* Entry 'Default': '<S680>:1' *)
                        (* '<S680>:1:2' BattSelect=0; *)
                        BattSelect := 0.0;
                    ELSE 
                        (* '<S680>:4:2' BattSelect = 2; *)
                        BattSelect := 2.0;
                    END_IF;

            END_CASE;

        END_IF;

        (* End of Chart: '<S675>/ChartBatt3' *)
END_CASE;

END_FUNCTION_BLOCK

// Device/Application/Lib_InputProcessing_state
FUNCTION_BLOCK Lib_InputProcessing_state
VAR_INPUT
	ssMethodType: SINT;
	Timeout: BOOL;
	Data_In: USINT;
END_VAR
VAR_OUTPUT
	u8Data_Out: USINT;
END_VAR
VAR
	Lib_InputProcessing_state_MODE: BOOL;
END_VAR



CASE ssMethodType OF
    SS_INITIALIZE: 
        (* SystemInitialize for Outport: '<S481>/u8Data_Out' *)
        u8Data_Out := 0;
    SS_OUTPUT: 
        (* Outputs for Enabled SubSystem: '<S428>/Lib_InputProcessing_state' incorporates:
         *  EnablePort: '<S481>/Timeout' *)

        IF Timeout THEN 

            IF  NOT Lib_InputProcessing_state_MODE THEN 
                Lib_InputProcessing_state_MODE := TRUE;
            END_IF;

            (* DataTypeConversion: '<S481>/Data Type Conversion' *)
            u8Data_Out := Data_In;
        ELSIF Lib_InputProcessing_state_MODE THEN 
            (* Disable for Outport: '<S481>/u8Data_Out' *)
            u8Data_Out := 0;
            Lib_InputProcessing_state_MODE := FALSE;
        END_IF;

        (* End of Outputs for SubSystem: '<S428>/Lib_InputProcessing_state' *)
    SS_DISABLE: 
        (* Disable for Outport: '<S481>/u8Data_Out' *)
        u8Data_Out := 0;
        Lib_InputProcessing_state_MODE := FALSE;
END_CASE;

END_FUNCTION_BLOCK

// Device/Application/IMD_OK
FUNCTION_BLOCK IMD_OK
VAR_INPUT
	ssMethodType: SINT;
	IP_boBMS_InsulationReadyOK: BOOL;
	Req_IMD: BOOL;
	IT_u8IMD_DelayTime_s_g: USINT;
END_VAR
VAR_OUTPUT
	IMD_OK_i: BOOL;
END_VAR
VAR
	temporalCounter_i1: PLC_CODER_TIMER;
	is_c63_ChiefMaster: USINT;
	is_active_c63_ChiefMaster: USINT;
	Req_IMD_prev: BOOL;
	Req_IMD_start: BOOL;
END_VAR



CASE ssMethodType OF
    SS_INITIALIZE: 
        temporalCounter_i1(timerAction := 1, maxTime := 0);
        is_active_c63_ChiefMaster := 0;
        is_c63_ChiefMaster := ChiefMaster_IN_NO_ACTIVE_CHILD_gd;
        IMD_OK_i := FALSE;
    SS_OUTPUT: 
        (* Gateway: ChiefMaster/Input Translation/Battery Signals/Subsystem7/Subsystem1/IMD_OK *)
        Req_IMD_prev := Req_IMD_start;
        Req_IMD_start := Req_IMD;
        (* Chart: '<S766>/IMD_OK' *)
        (* During: ChiefMaster/Input Translation/Battery Signals/Subsystem7/Subsystem1/IMD_OK *)

        IF is_active_c63_ChiefMaster = 0 THEN 
            Req_IMD_prev := Req_IMD;
            (* Entry: ChiefMaster/Input Translation/Battery Signals/Subsystem7/Subsystem1/IMD_OK *)
            is_active_c63_ChiefMaster := 1;
            (* Entry Internal: ChiefMaster/Input Translation/Battery Signals/Subsystem7/Subsystem1/IMD_OK *)
            (* Transition: '<S769>:3' *)
            is_c63_ChiefMaster := ChiefMaster_IN_Default_i;
            (* Entry 'Default': '<S769>:2' *)
            (* '<S769>:2:2' IMD_OK=false; *)
            IMD_OK_i := FALSE;
        ELSE 

            CASE is_c63_ChiefMaster OF
                ChiefMaster_IN_Default_i: 
                    (* During 'Default': '<S769>:2' *)
                    (* '<S769>:5:1' sf_internal_predicateOutput = IP_boBMS_InsulationReadyOK == true; *)

                    IF IP_boBMS_InsulationReadyOK THEN 
                        (* Transition: '<S769>:5' *)
                        is_c63_ChiefMaster := ChiefMaster_IN_Hold3;
                        temporalCounter_i1(timerAction := 1, maxTime := 0);
                        (* Entry 'Hold3': '<S769>:23' *)
                        (* '<S769>:23:2' IMD_OK=false; *)
                        IMD_OK_i := FALSE;
                    ELSE 
                        (* '<S769>:2:2' IMD_OK=false; *)
                        IMD_OK_i := FALSE;
                    END_IF;

                ChiefMaster_IN_Hold_m: 
                    (* During 'Hold': '<S769>:4' *)
                    (* '<S769>:19:1' sf_internal_predicateOutput = Req_IMD == false; *)

                    IF  NOT Req_IMD THEN 
                        (* Transition: '<S769>:19' *)
                        is_c63_ChiefMaster := ChiefMaster_IN_Hold2;
                        (* Entry 'Hold2': '<S769>:18' *)
                        (* '<S769>:18:2' IMD_OK=true; *)
                        IMD_OK_i := TRUE;
                    ELSE 
                        (* '<S769>:4:2' IMD_OK=true; *)
                        IMD_OK_i := TRUE;
                    END_IF;

                ChiefMaster_IN_Hold2: 
                    (* During 'Hold2': '<S769>:18' *)
                    (* '<S769>:13:1' sf_internal_predicateOutput = hasChangedFrom(Req_IMD,false); *)

                    IF (Req_IMD_prev <> Req_IMD_start) AND ( NOT Req_IMD_prev) THEN 
                        (* Transition: '<S769>:13' *)
                        (* Transition: '<S769>:26' *)
                        is_c63_ChiefMaster := ChiefMaster_IN_Default_i;
                        (* Entry 'Default': '<S769>:2' *)
                        (* '<S769>:2:2' IMD_OK=false; *)
                        IMD_OK_i := FALSE;
                    ELSE 
                        (* '<S769>:18:2' IMD_OK=true; *)
                        IMD_OK_i := TRUE;
                    END_IF;

                ELSE
                    (* During 'Hold3': '<S769>:23' *)
                    (* '<S769>:24:1' sf_internal_predicateOutput = after(IT_u8IMD_DelayTime_s,sec) &&... *)
                    (* '<S769>:24:2' IP_boBMS_InsulationReadyOK == true; *)
                    temporalCounter_i1(timerAction := 2, maxTime := USINT_TO_DINT(IT_u8IMD_DelayTime_s_g) * 1000);

                    IF temporalCounter_i1.done THEN 

                        IF IP_boBMS_InsulationReadyOK THEN 
                            (* Transition: '<S769>:24' *)
                            is_c63_ChiefMaster := ChiefMaster_IN_Hold_m;
                            (* Entry 'Hold': '<S769>:4' *)
                            (* '<S769>:4:2' IMD_OK=true; *)
                            IMD_OK_i := TRUE;
                        ELSE 
                            (* '<S769>:23:2' IMD_OK=false; *)
                            IMD_OK_i := FALSE;
                        END_IF;

                    ELSE 
                        (* '<S769>:23:2' IMD_OK=false; *)
                        IMD_OK_i := FALSE;
                    END_IF;

            END_CASE;

        END_IF;

        (* End of Chart: '<S766>/IMD_OK' *)
END_CASE;

END_FUNCTION_BLOCK

// Device/Application/REQ_HV_ON_Batt
FUNCTION_BLOCK REQ_HV_ON_Batt
VAR_INPUT
	ssMethodType: SINT;
	IsolationMeasurementRequest: BOOL;
	IP_boChargeStop_Pressed: BOOL;
	SafeToSD_BB1: BOOL;
	SafeToSD_BB2: BOOL;
	SafeToSD_BB3: BOOL;
	KL15_CM_disable: BOOL;
	SDError_BB1: BOOL;
	SDError_BB2: BOOL;
	SDError_BB3: BOOL;
	InsulationReadyOK_B1: BOOL;
	InsulationReadyOK_B2: BOOL;
	InsulationReadyOK_B3: BOOL;
	IMD_Active_BB1: BOOL;
	IMD_Active_BB2: BOOL;
	IMD_Active_BB3: BOOL;
	Software_Reset_KL15_BB3: LREAL;
	Software_Reset_KL15_BB2: LREAL;
	Software_Reset_KL15_BB1: LREAL;
	FL_boSafeToCloseHV_BB1: BOOL;
	FL_boSafeToCloseHV_BB2: BOOL;
	FL_boSafeToCloseHV_BB3: BOOL;
	FL_boST_REQ_HV_Open_BB1: BOOL;
	FL_boST_REQ_HV_Open_BB2: BOOL;
	FL_boST_REQ_HV_Open_BB3: BOOL;
	FL_boSystem_SD: BOOL;
	HV_Minus_Sense_BB1: BOOL;
	HV_Plus_Sense_BB1: BOOL;
	HV_Minus_Sense_BB2: BOOL;
	HV_Plus_Sense_BB2: BOOL;
	HV_Minus_Sense_BB3: BOOL;
	HV_Plus_Sense_BB3: BOOL;
	HV_REL_ON_BB2: BOOL;
	HV_REL_ON_BB1: BOOL;
	HV_REL_ON_BB3: BOOL;
	FL_boMainHV_SD_OK: BOOL;
	FL_boMainHV_PlusMinus_Status: BOOL;
END_VAR
VAR_OUTPUT
	FL_u8ContactorState_BB1: LREAL;
	FL_u8ContactorState_BB2: LREAL;
	FL_u8ContactorState_BB3: LREAL;
	FL_boREQ_HV_ON_BB1: LREAL;
	FL_boREQ_HV_ON_BB2: LREAL;
	FL_boREQ_HV_ON_BB3: LREAL;
	FL_u8Contactor_FB_State_BB1: LREAL;
	FL_u8Contactor_FB_State_BB2: LREAL;
	FL_u8Contactor_FB_State_BB3: LREAL;
END_VAR
VAR
	i0_Chart_REQ_HV_ON_Batt1: Chart_REQ_HV_ON_Batt1;
	i0_Chart_ContactorFB_State_Batt1: Chart_ContactorFB_State_Batt1;
	i0_Chart_REQ_HV_ON_Batt2: Chart_REQ_HV_ON_Batt2;
	i0_Chart_ContactorFB_State_Batt2: Chart_ContactorFB_State_Batt2;
	i0_Chart_REQ_HV_ON_Batt3: Chart_REQ_HV_ON_Batt3;
	i0_Chart_ContactorFB_State_Batt3: Chart_ContactorFB_State_Batt3;
END_VAR



CASE ssMethodType OF
    SS_INITIALIZE: 
        i0_Chart_REQ_HV_ON_Batt1(ssMethodType := SS_INITIALIZE, IP_boChargeStop_Pressed := IP_boChargeStop_Pressed, InsulationReadyOK := InsulationReadyOK_B1, SDError_BB := SDError_BB1, IMD_Active_BB1 := IMD_Active_BB1, IMD_Active_BB2 := IMD_Active_BB2, IMD_Active_BB3 := IMD_Active_BB3, Software_Reset_KL15_BB := Software_Reset_KL15_BB1, KL15_CM_disable := KL15_CM_disable, SafeToCloseHV_n := FL_boSafeToCloseHV_BB1, MainHV_SD_OK := FL_boMainHV_SD_OK, SafeToSD := SafeToSD_BB1, HV_REL_ON_BB2 := HV_REL_ON_BB2, HV_REL_ON_BB3 := HV_REL_ON_BB3, System_SD := FL_boSystem_SD, HV_REL_ON_BB1 := HV_REL_ON_BB1, MainHV_PlusMinus_Status := FL_boMainHV_PlusMinus_Status, IsolationMeasurementRequest := IsolationMeasurementRequest, REQ_HV_Open := FL_boST_REQ_HV_Open_BB1);
        FL_boREQ_HV_ON_BB1 := i0_Chart_REQ_HV_ON_Batt1.REQ_HV_ON;
        FL_u8ContactorState_BB1 := i0_Chart_REQ_HV_ON_Batt1.ContactorState;
        i0_Chart_ContactorFB_State_Batt1(ssMethodType := SS_INITIALIZE, HV_Minus_Sense_BB := HV_Minus_Sense_BB1, HV_Plus_Sense_BB := HV_Plus_Sense_BB1, REQ_HV_ON := FL_boREQ_HV_ON_BB1);
        FL_u8Contactor_FB_State_BB1 := i0_Chart_ContactorFB_State_Batt1.Contactor_FB_State;
        i0_Chart_REQ_HV_ON_Batt2(ssMethodType := SS_INITIALIZE, IP_boChargeStop_Pressed := IP_boChargeStop_Pressed, InsulationReadyOK := InsulationReadyOK_B2, SDError_BB := SDError_BB2, IMD_Active_BB1 := IMD_Active_BB1, IMD_Active_BB2 := IMD_Active_BB2, IMD_Active_BB3 := IMD_Active_BB3, Software_Reset_KL15_BB := Software_Reset_KL15_BB2, KL15_CM_disable := KL15_CM_disable, SafeToCloseHV_f := FL_boSafeToCloseHV_BB2, MainHV_SD_OK := FL_boMainHV_SD_OK, SafeToSD := SafeToSD_BB2, HV_REL_ON_BB1 := HV_REL_ON_BB1, HV_REL_ON_BB3 := HV_REL_ON_BB3, System_SD := FL_boSystem_SD, HV_REL_ON_BB2 := HV_REL_ON_BB2, MainHV_PlusMinus_Status := FL_boMainHV_PlusMinus_Status, IsolationMeasurementRequest := IsolationMeasurementRequest, REQ_HV_Open := FL_boST_REQ_HV_Open_BB2);
        FL_boREQ_HV_ON_BB2 := i0_Chart_REQ_HV_ON_Batt2.REQ_HV_ON;
        FL_u8ContactorState_BB2 := i0_Chart_REQ_HV_ON_Batt2.ContactorState;
        i0_Chart_ContactorFB_State_Batt2(ssMethodType := SS_INITIALIZE, HV_Minus_Sense_BB := HV_Minus_Sense_BB2, HV_Plus_Sense_BB := HV_Plus_Sense_BB2, REQ_HV_ON := FL_boREQ_HV_ON_BB2);
        FL_u8Contactor_FB_State_BB2 := i0_Chart_ContactorFB_State_Batt2.Contactor_FB_State;
        i0_Chart_REQ_HV_ON_Batt3(ssMethodType := SS_INITIALIZE, IP_boChargeStop_Pressed := IP_boChargeStop_Pressed, InsulationReadyOK := InsulationReadyOK_B3, SDError_BB := SDError_BB3, IMD_Active_BB1 := IMD_Active_BB1, IMD_Active_BB2 := IMD_Active_BB2, IMD_Active_BB3 := IMD_Active_BB3, Software_Reset_KL15_BB := Software_Reset_KL15_BB3, KL15_CM_disable := KL15_CM_disable, SafeToCloseHV_n := FL_boSafeToCloseHV_BB3, MainHV_SD_OK := FL_boMainHV_SD_OK, SafeToSD := SafeToSD_BB3, HV_REL_ON_BB1 := HV_REL_ON_BB1, HV_REL_ON_BB2 := HV_REL_ON_BB2, System_SD := FL_boSystem_SD, HV_REL_ON_BB3 := HV_REL_ON_BB3, MainHV_PlusMinus_Status := FL_boMainHV_PlusMinus_Status, IsolationMeasurementRequest := IsolationMeasurementRequest, REQ_HV_Open := FL_boST_REQ_HV_Open_BB3);
        FL_boREQ_HV_ON_BB3 := i0_Chart_REQ_HV_ON_Batt3.REQ_HV_ON;
        FL_u8ContactorState_BB3 := i0_Chart_REQ_HV_ON_Batt3.ContactorState;
        i0_Chart_ContactorFB_State_Batt3(ssMethodType := SS_INITIALIZE, HV_Minus_Sense_BB := HV_Minus_Sense_BB3, HV_Plus_Sense_BB := HV_Plus_Sense_BB3, REQ_HV_ON := FL_boREQ_HV_ON_BB3);
        FL_u8Contactor_FB_State_BB3 := i0_Chart_ContactorFB_State_Batt3.Contactor_FB_State;
    SS_OUTPUT: 
        i0_Chart_REQ_HV_ON_Batt1(ssMethodType := SS_OUTPUT, IP_boChargeStop_Pressed := IP_boChargeStop_Pressed, InsulationReadyOK := InsulationReadyOK_B1, SDError_BB := SDError_BB1, IMD_Active_BB1 := IMD_Active_BB1, IMD_Active_BB2 := IMD_Active_BB2, IMD_Active_BB3 := IMD_Active_BB3, Software_Reset_KL15_BB := Software_Reset_KL15_BB1, KL15_CM_disable := KL15_CM_disable, SafeToCloseHV_n := FL_boSafeToCloseHV_BB1, MainHV_SD_OK := FL_boMainHV_SD_OK, SafeToSD := SafeToSD_BB1, HV_REL_ON_BB2 := HV_REL_ON_BB2, HV_REL_ON_BB3 := HV_REL_ON_BB3, System_SD := FL_boSystem_SD, HV_REL_ON_BB1 := HV_REL_ON_BB1, MainHV_PlusMinus_Status := FL_boMainHV_PlusMinus_Status, IsolationMeasurementRequest := IsolationMeasurementRequest, REQ_HV_Open := FL_boST_REQ_HV_Open_BB1);
        FL_boREQ_HV_ON_BB1 := i0_Chart_REQ_HV_ON_Batt1.REQ_HV_ON;
        FL_u8ContactorState_BB1 := i0_Chart_REQ_HV_ON_Batt1.ContactorState;
        i0_Chart_ContactorFB_State_Batt1(ssMethodType := SS_OUTPUT, HV_Minus_Sense_BB := HV_Minus_Sense_BB1, HV_Plus_Sense_BB := HV_Plus_Sense_BB1, REQ_HV_ON := FL_boREQ_HV_ON_BB1);
        FL_u8Contactor_FB_State_BB1 := i0_Chart_ContactorFB_State_Batt1.Contactor_FB_State;
        i0_Chart_REQ_HV_ON_Batt2(ssMethodType := SS_OUTPUT, IP_boChargeStop_Pressed := IP_boChargeStop_Pressed, InsulationReadyOK := InsulationReadyOK_B2, SDError_BB := SDError_BB2, IMD_Active_BB1 := IMD_Active_BB1, IMD_Active_BB2 := IMD_Active_BB2, IMD_Active_BB3 := IMD_Active_BB3, Software_Reset_KL15_BB := Software_Reset_KL15_BB2, KL15_CM_disable := KL15_CM_disable, SafeToCloseHV_f := FL_boSafeToCloseHV_BB2, MainHV_SD_OK := FL_boMainHV_SD_OK, SafeToSD := SafeToSD_BB2, HV_REL_ON_BB1 := HV_REL_ON_BB1, HV_REL_ON_BB3 := HV_REL_ON_BB3, System_SD := FL_boSystem_SD, HV_REL_ON_BB2 := HV_REL_ON_BB2, MainHV_PlusMinus_Status := FL_boMainHV_PlusMinus_Status, IsolationMeasurementRequest := IsolationMeasurementRequest, REQ_HV_Open := FL_boST_REQ_HV_Open_BB2);
        FL_boREQ_HV_ON_BB2 := i0_Chart_REQ_HV_ON_Batt2.REQ_HV_ON;
        FL_u8ContactorState_BB2 := i0_Chart_REQ_HV_ON_Batt2.ContactorState;
        i0_Chart_ContactorFB_State_Batt2(ssMethodType := SS_OUTPUT, HV_Minus_Sense_BB := HV_Minus_Sense_BB2, HV_Plus_Sense_BB := HV_Plus_Sense_BB2, REQ_HV_ON := FL_boREQ_HV_ON_BB2);
        FL_u8Contactor_FB_State_BB2 := i0_Chart_ContactorFB_State_Batt2.Contactor_FB_State;
        i0_Chart_REQ_HV_ON_Batt3(ssMethodType := SS_OUTPUT, IP_boChargeStop_Pressed := IP_boChargeStop_Pressed, InsulationReadyOK := InsulationReadyOK_B3, SDError_BB := SDError_BB3, IMD_Active_BB1 := IMD_Active_BB1, IMD_Active_BB2 := IMD_Active_BB2, IMD_Active_BB3 := IMD_Active_BB3, Software_Reset_KL15_BB := Software_Reset_KL15_BB3, KL15_CM_disable := KL15_CM_disable, SafeToCloseHV_n := FL_boSafeToCloseHV_BB3, MainHV_SD_OK := FL_boMainHV_SD_OK, SafeToSD := SafeToSD_BB3, HV_REL_ON_BB1 := HV_REL_ON_BB1, HV_REL_ON_BB2 := HV_REL_ON_BB2, System_SD := FL_boSystem_SD, HV_REL_ON_BB3 := HV_REL_ON_BB3, MainHV_PlusMinus_Status := FL_boMainHV_PlusMinus_Status, IsolationMeasurementRequest := IsolationMeasurementRequest, REQ_HV_Open := FL_boST_REQ_HV_Open_BB3);
        FL_boREQ_HV_ON_BB3 := i0_Chart_REQ_HV_ON_Batt3.REQ_HV_ON;
        FL_u8ContactorState_BB3 := i0_Chart_REQ_HV_ON_Batt3.ContactorState;
        i0_Chart_ContactorFB_State_Batt3(ssMethodType := SS_OUTPUT, HV_Minus_Sense_BB := HV_Minus_Sense_BB3, HV_Plus_Sense_BB := HV_Plus_Sense_BB3, REQ_HV_ON := FL_boREQ_HV_ON_BB3);
        FL_u8Contactor_FB_State_BB3 := i0_Chart_ContactorFB_State_Batt3.Contactor_FB_State;
END_CASE;

END_FUNCTION_BLOCK

// Device/Application/Chart_REQ_HV_ON_Batt1
FUNCTION_BLOCK Chart_REQ_HV_ON_Batt1
VAR_INPUT
	ssMethodType: SINT;
	IP_boChargeStop_Pressed: BOOL;
	InsulationReadyOK: BOOL;
	SDError_BB: BOOL;
	IMD_Active_BB1: BOOL;
	IMD_Active_BB2: BOOL;
	IMD_Active_BB3: BOOL;
	Software_Reset_KL15_BB: LREAL;
	KL15_CM_disable: BOOL;
	SafeToCloseHV_n: BOOL;
	MainHV_SD_OK: BOOL;
	SafeToSD: BOOL;
	HV_REL_ON_BB2: BOOL;
	HV_REL_ON_BB3: BOOL;
	System_SD: BOOL;
	HV_REL_ON_BB1: BOOL;
	MainHV_PlusMinus_Status: BOOL;
	IsolationMeasurementRequest: BOOL;
	REQ_HV_Open: BOOL;
END_VAR
VAR_OUTPUT
	REQ_HV_ON: LREAL;
	ContactorState: LREAL;
END_VAR
VAR
	temporalCounter_i1: PLC_CODER_TIMER;
	temporalCounter_i2: PLC_CODER_TIMER;
	is_c1_ChiefMaster: USINT;
	is_active_c1_ChiefMaster: USINT;
	tmp: BOOL;
	temp1: BOOL;
	temp2: BOOL;
	temp3: BOOL;
	temp4: BOOL;
	temp5: BOOL;
END_VAR



CASE ssMethodType OF
    SS_INITIALIZE: 
        temporalCounter_i1(timerAction := 1, maxTime := 0);
        temporalCounter_i2(timerAction := 1, maxTime := 0);
        temporalCounter_i1(timerAction := 1, maxTime := 0);
        is_active_c1_ChiefMaster := 0;
        is_c1_ChiefMaster := ChiefMaster_IN_NO_ACTIVE_CHILD_d;
        REQ_HV_ON := 0.0;
        ContactorState := 0.0;
    SS_OUTPUT: 
        (* Chart: '<S33>/Chart_REQ_HV_ON_Batt1' *)
        (* Gateway: ChiefMaster/Flow Logic/Battery HVControl/REQ_HV_ON_Batt/Chart_REQ_HV_ON_Batt1 *)
        (* During: ChiefMaster/Flow Logic/Battery HVControl/REQ_HV_ON_Batt/Chart_REQ_HV_ON_Batt1 *)

        IF is_active_c1_ChiefMaster = 0 THEN 
            (* Entry: ChiefMaster/Flow Logic/Battery HVControl/REQ_HV_ON_Batt/Chart_REQ_HV_ON_Batt1 *)
            is_active_c1_ChiefMaster := 1;
            (* Entry Internal: ChiefMaster/Flow Logic/Battery HVControl/REQ_HV_ON_Batt/Chart_REQ_HV_ON_Batt1 *)
            (* Transition: '<S40>:8' *)
            is_c1_ChiefMaster := b_ChiefMaster_IN_Default_h;
            (* Entry 'Default': '<S40>:7' *)
            (* '<S40>:7:2' REQ_HV_ON = 0 *)
            REQ_HV_ON := 0.0;
            (* '<S40>:7:3' ContactorState = 1 *)
            ContactorState := 1.0;
        ELSE 
            temp2 := FALSE;
            temp3 := FALSE;
            temp4 := FALSE;
            temp5 := FALSE;

            CASE is_c1_ChiefMaster OF
                ChiefMaster_IN_CONTACTOR_OFF: 
                    (* During 'CONTACTOR_OFF': '<S40>:18' *)
                    (* '<S40>:23:1' sf_internal_predicateOutput = InsulationReadyOK == false ||... *)
                    (* '<S40>:23:2' SDError_BB == true ||... *)
                    (* '<S40>:23:3' Software_Reset_KL15_BB == true ||... *)
                    (* '<S40>:23:4' KL15_CM_disable == true; *)

                    IF ((( NOT InsulationReadyOK) OR SDError_BB) OR (Software_Reset_KL15_BB = 1.0)) OR KL15_CM_disable THEN 
                        (* Transition: '<S40>:23' *)
                        is_c1_ChiefMaster := b_ChiefMaster_IN_Default_h;
                        (* Entry 'Default': '<S40>:7' *)
                        (* '<S40>:7:2' REQ_HV_ON = 0 *)
                        REQ_HV_ON := 0.0;
                        (* '<S40>:7:3' ContactorState = 1 *)
                        ContactorState := 1.0;
                    ELSE 
                        (* '<S40>:21:1' sf_internal_predicateOutput = after(2,sec) &&... *)
                        (* '<S40>:21:2' IMD_Active_BB1 == true &&... *)
                        (* '<S40>:21:3' IMD_Active_BB2 == false &&... *)
                        (* '<S40>:21:4' IMD_Active_BB3 == false &&... *)
                        (* '<S40>:21:5' MainHV_PlusMinus_Status == 0; *)
                        temporalCounter_i1(timerAction := 2, maxTime := 2000);

                        IF temporalCounter_i1.done THEN 

                            IF ((IMD_Active_BB1 AND ( NOT IMD_Active_BB2)) AND ( NOT IMD_Active_BB3)) AND ( NOT MainHV_PlusMinus_Status) THEN 
                                (* Transition: '<S40>:21' *)
                                temp3 := TRUE;
                            ELSE 
                                temp5 := TRUE;
                            END_IF;

                        ELSE 
                            temp5 := TRUE;
                        END_IF;

                    END_IF;

                ChiefMaster_IN_CONTACTOR_ON: 
                    (* During 'CONTACTOR_ON': '<S40>:20' *)
                    (* '<S40>:44:1' sf_internal_predicateOutput = (KL15_CM_disable == true || System_SD == true || SDError_BB == true) &&... *)
                    (* '<S40>:44:2' (MainHV_SD_OK == true || HV_REL_ON_BB1 == false); *)
                    tmp :=  NOT HV_REL_ON_BB1;

                    IF ((KL15_CM_disable OR System_SD) OR SDError_BB) AND (MainHV_SD_OK OR tmp) THEN 
                        (* Transition: '<S40>:44' *)
                        is_c1_ChiefMaster := ChiefMaster_IN_hold_hp;
                        temporalCounter_i1(timerAction := 1, maxTime := 0);
                    ELSE 
                        (* '<S40>:51:1' sf_internal_predicateOutput = SDError_BB == true &&... *)
                        (* '<S40>:51:2' (HV_REL_ON_BB2 == true || HV_REL_ON_BB3 == true) &&... *)
                        (* '<S40>:51:3' (SafeToSD == true || HV_REL_ON_BB1 == false); *)
                        temp1 := HV_REL_ON_BB2 OR HV_REL_ON_BB3;

                        IF (SDError_BB AND temp1) AND (SafeToSD OR tmp) THEN 
                            (* Transition: '<S40>:51' *)
                            temp4 := TRUE;
                        ELSE 
                            (* '<S40>:68:1' sf_internal_predicateOutput = (HV_REL_ON_BB2 == true || HV_REL_ON_BB3 == true) &&... *)
                            (* '<S40>:68:2' REQ_HV_Open == true; *)

                            IF temp1 AND REQ_HV_Open THEN 
                                (* Transition: '<S40>:68' *)
                                temp4 := TRUE;
                            ELSE 
                                (* '<S40>:20:2' REQ_HV_ON = 1 *)
                                REQ_HV_ON := 1.0;
                                (* '<S40>:20:3' ContactorState = 3 *)
                                ContactorState := 3.0;
                            END_IF;

                        END_IF;

                    END_IF;

                b_ChiefMaster_IN_Default_h: 
                    (* During 'Default': '<S40>:7' *)
                    (* '<S40>:19:1' sf_internal_predicateOutput = IP_boChargeStop_Pressed == false &&... *)
                    (* '<S40>:19:2' KL15_CM_disable == false &&... *)
                    (* '<S40>:19:3' InsulationReadyOK == true &&... *)
                    (* '<S40>:19:4' SDError_BB == false &&... *)
                    (* '<S40>:19:5' System_SD == false; *)

                    IF (((( NOT IP_boChargeStop_Pressed) AND ( NOT KL15_CM_disable)) AND InsulationReadyOK) AND ( NOT SDError_BB)) AND ( NOT System_SD) THEN 
                        (* Transition: '<S40>:19' *)
                        is_c1_ChiefMaster := ChiefMaster_IN_CONTACTOR_OFF;
                        temporalCounter_i1(timerAction := 1, maxTime := 0);
                        temporalCounter_i2(timerAction := 1, maxTime := 0);
                        (* Entry 'CONTACTOR_OFF': '<S40>:18' *)
                        (* '<S40>:18:2' REQ_HV_ON = 0 *)
                        REQ_HV_ON := 0.0;
                        (* '<S40>:18:3' ContactorState = 2 *)
                        ContactorState := 2.0;
                    ELSE 
                        (* '<S40>:7:2' REQ_HV_ON = 0 *)
                        REQ_HV_ON := 0.0;
                        (* '<S40>:7:3' ContactorState = 1 *)
                        ContactorState := 1.0;
                    END_IF;

                ELSE
                    (* During 'hold': '<S40>:64' *)
                    (* '<S40>:65:1' sf_internal_predicateOutput = after(2,sec); *)
                    temporalCounter_i1(timerAction := 2, maxTime := 2000);

                    IF temporalCounter_i1.done THEN 
                        (* Transition: '<S40>:65' *)
                        is_c1_ChiefMaster := b_ChiefMaster_IN_Default_h;
                        (* Entry 'Default': '<S40>:7' *)
                        (* '<S40>:7:2' REQ_HV_ON = 0 *)
                        REQ_HV_ON := 0.0;
                        (* '<S40>:7:3' ContactorState = 1 *)
                        ContactorState := 1.0;
                    END_IF;

            END_CASE;


            IF temp5 THEN 
                (* '<S40>:28:1' sf_internal_predicateOutput = after(2,sec) &&... *)
                (* '<S40>:28:2' IMD_Active_BB1 == false &&... *)
                (* '<S40>:28:3' MainHV_PlusMinus_Status == 1 &&... *)
                (* '<S40>:28:4' (IMD_Active_BB2 == true || IMD_Active_BB3 ==true || IsolationMeasurementRequest == false) &&... *)
                (* '<S40>:28:5' SafeToCloseHV == true; *)
                temporalCounter_i2(timerAction := 2, maxTime := 2000);

                IF temporalCounter_i2.done THEN 

                    IF ((( NOT IMD_Active_BB1) AND MainHV_PlusMinus_Status) AND ((IMD_Active_BB2 OR IMD_Active_BB3) OR ( NOT IsolationMeasurementRequest))) AND SafeToCloseHV_n THEN 
                        (* Transition: '<S40>:28' *)
                        temp3 := TRUE;
                    ELSE 
                        temp2 := TRUE;
                    END_IF;

                ELSE 
                    temp2 := TRUE;
                END_IF;

            END_IF;


            IF temp4 THEN 
                is_c1_ChiefMaster := b_ChiefMaster_IN_Default_h;
                (* Entry 'Default': '<S40>:7' *)
                (* '<S40>:7:2' REQ_HV_ON = 0 *)
                REQ_HV_ON := 0.0;
                (* '<S40>:7:3' ContactorState = 1 *)
                ContactorState := 1.0;
            END_IF;


            IF temp3 THEN 
                is_c1_ChiefMaster := ChiefMaster_IN_CONTACTOR_ON;
                (* Entry 'CONTACTOR_ON': '<S40>:20' *)
                (* '<S40>:20:2' REQ_HV_ON = 1 *)
                REQ_HV_ON := 1.0;
                (* '<S40>:20:3' ContactorState = 3 *)
                ContactorState := 3.0;
            END_IF;


            IF temp2 THEN 
                (* '<S40>:18:2' REQ_HV_ON = 0 *)
                REQ_HV_ON := 0.0;
                (* '<S40>:18:3' ContactorState = 2 *)
                ContactorState := 2.0;
            END_IF;

        END_IF;

        (* End of Chart: '<S33>/Chart_REQ_HV_ON_Batt1' *)
END_CASE;

END_FUNCTION_BLOCK

// Device/Application/SafeToCloseHV
FUNCTION_BLOCK SafeToCloseHV
VAR_INPUT
	FL_sVtgExt_BB1: REAL;
	FL_sVtgExt_BB2: REAL;
	FL_sVtgExt_BB3: REAL;
	VtgInt_BB1: REAL;
	VtgInt_BB2: REAL;
	VtgInt_BB3: REAL;
	IMD_Active_BB1: BOOL;
	IMD_Active_BB2: BOOL;
	IMD_Active_BB3: BOOL;
	InternalResistance_BB1: REAL;
	InternalResistance_BB2: REAL;
	InternalResistance_BB3: REAL;
	HV_REL_ON_BB1: BOOL;
	HV_REL_ON_BB2: BOOL;
	HV_REL_ON_BB3: BOOL;
END_VAR
VAR_OUTPUT
	FL_boSafeToCloseHV_BB1: BOOL;
	FL_boSafeToCloseHV_BB2: BOOL;
	FL_boSafeToCloseHV_BB3: BOOL;
	FL_sCalculated_Vtg_Diff_BB1: REAL;
	FL_sCalculated_Vtg_Diff_BB2: REAL;
	FL_sCalculated_Vtg_Diff_BB3: REAL;
	FL_sCalculated_InrushCurrent_BB1: REAL;
	FL_sCalculated_InrushCurrent_BB2: REAL;
	FL_sCalculated_InrushCurrent_BB3: REAL;
END_VAR
VAR
	rtb_Add1_h: REAL;
	rtb_Add2_a: REAL;
	temp1: REAL;
	temp2: REAL;
	temp3: REAL;
	temp6: REAL;
END_VAR


(* Switch: '<S34>/Switch' incorporates:
 *  Switch: '<S34>/Switch1'
 *  Switch: '<S34>/Switch2' *)

IF IMD_Active_BB1 THEN 
    FL_sCalculated_Vtg_Diff_BB3 := FL_sVtgExt_BB1;
ELSIF IMD_Active_BB2 THEN 
    (* Switch: '<S34>/Switch1' *)
    FL_sCalculated_Vtg_Diff_BB3 := FL_sVtgExt_BB2;
ELSIF IMD_Active_BB3 THEN 
    (* Switch: '<S34>/Switch2' incorporates:
     *  Switch: '<S34>/Switch1' *)
    FL_sCalculated_Vtg_Diff_BB3 := FL_sVtgExt_BB3;
ELSE 
    (* Switch: '<S34>/Switch2' incorporates:
     *  MinMax: '<S34>/Min'
     *  Product: '<S34>/Product3'
     *  Product: '<S34>/Product4'
     *  Product: '<S34>/Product5'
     *  Switch: '<S34>/Switch1' *)

    IF HV_REL_ON_BB1 THEN 
        temp1 := FL_sVtgExt_BB1;
    ELSE 
        temp1 := 0.0;
    END_IF;


    IF HV_REL_ON_BB2 THEN 
        temp2 := FL_sVtgExt_BB2;
    ELSE 
        temp2 := 0.0;
    END_IF;


    IF HV_REL_ON_BB3 THEN 
        temp3 := FL_sVtgExt_BB3;
    ELSE 
        temp3 := 0.0;
    END_IF;

    temp6 := MAX(temp1, temp2);
    FL_sCalculated_Vtg_Diff_BB3 := MAX(temp6, temp3);
END_IF;

(* End of Switch: '<S34>/Switch' *)


(* Abs: '<S34>/Abs' incorporates:
 *  Sum: '<S34>/Subtract' *)
FL_sCalculated_Vtg_Diff_BB1 := ABS(VtgInt_BB1 - FL_sCalculated_Vtg_Diff_BB3);
(* Abs: '<S34>/Abs1' incorporates:
 *  Sum: '<S34>/Subtract1' *)
FL_sCalculated_Vtg_Diff_BB2 := ABS(VtgInt_BB2 - FL_sCalculated_Vtg_Diff_BB3);
(* Sum: '<S34>/Subtract2' *)
FL_sCalculated_Vtg_Diff_BB3 := VtgInt_BB3 - FL_sCalculated_Vtg_Diff_BB3;
(* Abs: '<S34>/Abs2' *)
FL_sCalculated_Vtg_Diff_BB3 := ABS(FL_sCalculated_Vtg_Diff_BB3);
(* Product: '<S34>/Product' *)

IF HV_REL_ON_BB2 THEN 
    FL_sCalculated_InrushCurrent_BB3 := InternalResistance_BB2;
ELSE 
    FL_sCalculated_InrushCurrent_BB3 := 0.0;
END_IF;

(* Product: '<S34>/Product1' *)

IF HV_REL_ON_BB3 THEN 
    FL_sCalculated_InrushCurrent_BB2 := InternalResistance_BB3;
ELSE 
    FL_sCalculated_InrushCurrent_BB2 := 0.0;
END_IF;

(* Product: '<S34>/Product2' *)

IF HV_REL_ON_BB1 THEN 
    FL_sCalculated_InrushCurrent_BB1 := InternalResistance_BB1;
ELSE 
    FL_sCalculated_InrushCurrent_BB1 := 0.0;
END_IF;

(* Sum: '<S34>/Add1' *)
rtb_Add1_h := (FL_sCalculated_InrushCurrent_BB1 + FL_sCalculated_InrushCurrent_BB2) + InternalResistance_BB2;
(* Sum: '<S34>/Add2' *)
rtb_Add2_a := (FL_sCalculated_InrushCurrent_BB3 + FL_sCalculated_InrushCurrent_BB1) + InternalResistance_BB3;
(* Product: '<S34>/Divide' incorporates:
 *  Constant: '<S34>/Constant'
 *  Sum: '<S34>/Add'
 *  Sum: '<S34>/Add3' *)
FL_sCalculated_InrushCurrent_BB1 := FL_sCalculated_Vtg_Diff_BB1 / (((FL_sCalculated_InrushCurrent_BB3 + FL_sCalculated_InrushCurrent_BB2) + InternalResistance_BB1) + FL_sInrushCurrent_dividebyzero);
(* Product: '<S34>/Divide1' incorporates:
 *  Constant: '<S34>/Constant'
 *  Sum: '<S34>/Add4' *)
FL_sCalculated_InrushCurrent_BB2 := FL_sCalculated_Vtg_Diff_BB2 / (rtb_Add1_h + FL_sInrushCurrent_dividebyzero);
(* Product: '<S34>/Divide2' incorporates:
 *  Constant: '<S34>/Constant'
 *  Sum: '<S34>/Add5' *)
FL_sCalculated_InrushCurrent_BB3 := FL_sCalculated_Vtg_Diff_BB3 / (rtb_Add2_a + FL_sInrushCurrent_dividebyzero);
(* Logic: '<S34>/OR3' *)
FL_boSafeToCloseHV_BB3 := (HV_REL_ON_BB1 OR HV_REL_ON_BB2) OR HV_REL_ON_BB3;
(* Logic: '<S34>/OR' incorporates:
 *  Constant: '<S34>/SafeCurrentToCloseHV_A'
 *  Constant: '<S34>/SafeVoltageToCloseHV_V'
 *  Logic: '<S34>/OR4'
 *  RelationalOperator: '<S34>/Less Than'
 *  RelationalOperator: '<S34>/Less Than3' *)
FL_boSafeToCloseHV_BB1 := (FL_sCalculated_Vtg_Diff_BB1 < SafeVoltageToCloseHV_V) OR ((FL_sCalculated_InrushCurrent_BB1 < SafeCurrentToCloseHV_A) AND FL_boSafeToCloseHV_BB3);
(* Logic: '<S34>/OR1' incorporates:
 *  Constant: '<S34>/SafeCurrentToCloseHV_A'
 *  Constant: '<S34>/SafeVoltageToCloseHV_V'
 *  Logic: '<S34>/OR5'
 *  RelationalOperator: '<S34>/Less Than1'
 *  RelationalOperator: '<S34>/Less Than4' *)
FL_boSafeToCloseHV_BB2 := (FL_sCalculated_Vtg_Diff_BB2 < SafeVoltageToCloseHV_V) OR ((FL_sCalculated_InrushCurrent_BB2 < SafeCurrentToCloseHV_A) AND FL_boSafeToCloseHV_BB3);
(* Logic: '<S34>/OR2' incorporates:
 *  Constant: '<S34>/SafeCurrentToCloseHV_A'
 *  Constant: '<S34>/SafeVoltageToCloseHV_V'
 *  Logic: '<S34>/OR6'
 *  RelationalOperator: '<S34>/Less Than2'
 *  RelationalOperator: '<S34>/Less Than5' *)
FL_boSafeToCloseHV_BB3 := (FL_sCalculated_Vtg_Diff_BB3 < SafeVoltageToCloseHV_V) OR ((FL_sCalculated_InrushCurrent_BB3 < SafeCurrentToCloseHV_A) AND FL_boSafeToCloseHV_BB3);

END_FUNCTION_BLOCK

// Device/Application/Chart_ContactorFB_State_Batt1
FUNCTION_BLOCK Chart_ContactorFB_State_Batt1
VAR_INPUT
	ssMethodType: SINT;
	HV_Minus_Sense_BB: BOOL;
	HV_Plus_Sense_BB: BOOL;
	REQ_HV_ON: LREAL;
END_VAR
VAR_OUTPUT
	Contactor_FB_State: LREAL;
END_VAR
VAR
	temporalCounter_i1: PLC_CODER_TIMER;
	is_c37_ChiefMaster: USINT;
	is_active_c37_ChiefMaster: USINT;
END_VAR



CASE ssMethodType OF
    SS_INITIALIZE: 
        temporalCounter_i1(timerAction := 1, maxTime := 0);
        is_active_c37_ChiefMaster := 0;
        is_c37_ChiefMaster := ChiefMaster_IN_NO_ACTIVE_CHILD_m;
        Contactor_FB_State := 0.0;
    SS_OUTPUT: 
        (* Chart: '<S33>/Chart_ContactorFB_State_Batt1' *)
        (* Gateway: ChiefMaster/Flow Logic/Battery HVControl/REQ_HV_ON_Batt/Chart_ContactorFB_State_Batt1 *)
        (* During: ChiefMaster/Flow Logic/Battery HVControl/REQ_HV_ON_Batt/Chart_ContactorFB_State_Batt1 *)

        IF is_active_c37_ChiefMaster = 0 THEN 
            (* Entry: ChiefMaster/Flow Logic/Battery HVControl/REQ_HV_ON_Batt/Chart_ContactorFB_State_Batt1 *)
            is_active_c37_ChiefMaster := 1;
            (* Entry Internal: ChiefMaster/Flow Logic/Battery HVControl/REQ_HV_ON_Batt/Chart_ContactorFB_State_Batt1 *)
            (* Transition: '<S37>:2' *)
            is_c37_ChiefMaster := b_ChiefMaster_IN_default;
            (* Entry 'default': '<S37>:1' *)
            (* '<S37>:1:2' Contactor_FB_State = 0 *)
            Contactor_FB_State := 0.0;
        ELSE 

            CASE is_c37_ChiefMaster OF
                ChiefMaster_IN_Error_l: 
                    (* During 'Error': '<S37>:12' *)
                    (* '<S37>:51:1' sf_internal_predicateOutput = REQ_HV_ON == 1; *)

                    IF REQ_HV_ON = 1.0 THEN 
                        (* Transition: '<S37>:51' *)
                        is_c37_ChiefMaster := b_ChiefMaster_IN_default;
                        (* Entry 'default': '<S37>:1' *)
                        (* '<S37>:1:2' Contactor_FB_State = 0 *)
                        Contactor_FB_State := 0.0;
                    ELSE 
                        (* '<S37>:12:2' Contactor_FB_State = 3 *)
                        Contactor_FB_State := 3.0;
                    END_IF;

                ChiefMaster_IN_Open_m: 
                    (* During 'Open': '<S37>:46' *)
                    (* '<S37>:50:1' sf_internal_predicateOutput = REQ_HV_ON == 1; *)

                    IF REQ_HV_ON = 1.0 THEN 
                        (* Transition: '<S37>:50' *)
                        is_c37_ChiefMaster := b_ChiefMaster_IN_default;
                        (* Entry 'default': '<S37>:1' *)
                        (* '<S37>:1:2' Contactor_FB_State = 0 *)
                        Contactor_FB_State := 0.0;
                    ELSE 
                        (* '<S37>:46:2' Contactor_FB_State = 1 *)
                        Contactor_FB_State := 1.0;
                    END_IF;

                b_ChiefMaster_IN_default: 
                    (* During 'default': '<S37>:1' *)
                    (* '<S37>:5:1' sf_internal_predicateOutput = REQ_HV_ON == 0; *)

                    IF REQ_HV_ON = 0.0 THEN 
                        (* Transition: '<S37>:5' *)
                        is_c37_ChiefMaster := b_ChiefMaster_IN_hold;
                        temporalCounter_i1(timerAction := 1, maxTime := 0);
                        (* Entry 'hold': '<S37>:4' *)
                        (* '<S37>:4:2' Contactor_FB_State = 0 *)
                        Contactor_FB_State := 0.0;
                    ELSE 
                        (* '<S37>:1:2' Contactor_FB_State = 0 *)
                        Contactor_FB_State := 0.0;
                    END_IF;

                ELSE
                    (* During 'hold': '<S37>:4' *)
                    (* '<S37>:13:1' sf_internal_predicateOutput = after(5,sec); *)
                    temporalCounter_i1(timerAction := 2, maxTime := 5000);

                    IF temporalCounter_i1.done THEN 
                        (* Transition: '<S37>:13' *)
                        is_c37_ChiefMaster := ChiefMaster_IN_Error_l;
                        (* Entry 'Error': '<S37>:12' *)
                        (* '<S37>:12:2' Contactor_FB_State = 3 *)
                        Contactor_FB_State := 3.0;
                    ELSE 
                        (* '<S37>:47:1' sf_internal_predicateOutput = HV_Plus_Sense_BB == false &&... *)
                        (* '<S37>:47:2' HV_Minus_Sense_BB == false; *)

                        IF ( NOT HV_Plus_Sense_BB) AND ( NOT HV_Minus_Sense_BB) THEN 
                            (* Transition: '<S37>:47' *)
                            is_c37_ChiefMaster := ChiefMaster_IN_Open_m;
                            (* Entry 'Open': '<S37>:46' *)
                            (* '<S37>:46:2' Contactor_FB_State = 1 *)
                            Contactor_FB_State := 1.0;
                        ELSE 
                            (* '<S37>:4:2' Contactor_FB_State = 0 *)
                            Contactor_FB_State := 0.0;
                        END_IF;

                    END_IF;

            END_CASE;

        END_IF;

        (* End of Chart: '<S33>/Chart_ContactorFB_State_Batt1' *)
END_CASE;

END_FUNCTION_BLOCK

// Device/Application/Chart_REQ_HV_ON_Batt2
FUNCTION_BLOCK Chart_REQ_HV_ON_Batt2
VAR_INPUT
	ssMethodType: SINT;
	IP_boChargeStop_Pressed: BOOL;
	InsulationReadyOK: BOOL;
	SDError_BB: BOOL;
	IMD_Active_BB1: BOOL;
	IMD_Active_BB2: BOOL;
	IMD_Active_BB3: BOOL;
	Software_Reset_KL15_BB: LREAL;
	KL15_CM_disable: BOOL;
	SafeToCloseHV_f: BOOL;
	MainHV_SD_OK: BOOL;
	SafeToSD: BOOL;
	HV_REL_ON_BB1: BOOL;
	HV_REL_ON_BB3: BOOL;
	System_SD: BOOL;
	HV_REL_ON_BB2: BOOL;
	MainHV_PlusMinus_Status: BOOL;
	IsolationMeasurementRequest: BOOL;
	REQ_HV_Open: BOOL;
END_VAR
VAR_OUTPUT
	REQ_HV_ON: LREAL;
	ContactorState: LREAL;
END_VAR
VAR
	temporalCounter_i1: PLC_CODER_TIMER;
	temporalCounter_i2: PLC_CODER_TIMER;
	is_c5_ChiefMaster: USINT;
	is_active_c5_ChiefMaster: USINT;
	tmp: BOOL;
	temp1: BOOL;
	temp2: BOOL;
	temp3: BOOL;
	temp4: BOOL;
	temp5: BOOL;
END_VAR



CASE ssMethodType OF
    SS_INITIALIZE: 
        temporalCounter_i1(timerAction := 1, maxTime := 0);
        temporalCounter_i2(timerAction := 1, maxTime := 0);
        temporalCounter_i1(timerAction := 1, maxTime := 0);
        is_active_c5_ChiefMaster := 0;
        is_c5_ChiefMaster := ChiefMaster_IN_NO_ACTIVE_CHILD_iv;
        REQ_HV_ON := 0.0;
        ContactorState := 0.0;
    SS_OUTPUT: 
        (* Chart: '<S33>/Chart_REQ_HV_ON_Batt2 ' *)
        (* Gateway: ChiefMaster/Flow Logic/Battery HVControl/REQ_HV_ON_Batt/Chart_REQ_HV_ON_Batt2  *)
        (* During: ChiefMaster/Flow Logic/Battery HVControl/REQ_HV_ON_Batt/Chart_REQ_HV_ON_Batt2  *)

        IF is_active_c5_ChiefMaster = 0 THEN 
            (* Entry: ChiefMaster/Flow Logic/Battery HVControl/REQ_HV_ON_Batt/Chart_REQ_HV_ON_Batt2  *)
            is_active_c5_ChiefMaster := 1;
            (* Entry Internal: ChiefMaster/Flow Logic/Battery HVControl/REQ_HV_ON_Batt/Chart_REQ_HV_ON_Batt2  *)
            (* Transition: '<S41>:8' *)
            is_c5_ChiefMaster := b_ChiefMaster_IN_Default_n;
            (* Entry 'Default': '<S41>:7' *)
            (* '<S41>:7:2' REQ_HV_ON = 0 *)
            REQ_HV_ON := 0.0;
            (* '<S41>:7:3' ContactorState = 1 *)
            ContactorState := 1.0;
        ELSE 
            temp2 := FALSE;
            temp3 := FALSE;
            temp4 := FALSE;
            temp5 := FALSE;

            CASE is_c5_ChiefMaster OF
                ChiefMaster_IN_CONTACTOR_OFF_p: 
                    (* During 'CONTACTOR_OFF': '<S41>:18' *)
                    (* '<S41>:23:1' sf_internal_predicateOutput = InsulationReadyOK == false ||... *)
                    (* '<S41>:23:2' SDError_BB == true ||... *)
                    (* '<S41>:23:3' Software_Reset_KL15_BB == true ||... *)
                    (* '<S41>:23:4' KL15_CM_disable == true; *)

                    IF ((( NOT InsulationReadyOK) OR SDError_BB) OR (Software_Reset_KL15_BB = 1.0)) OR KL15_CM_disable THEN 
                        (* Transition: '<S41>:23' *)
                        is_c5_ChiefMaster := b_ChiefMaster_IN_Default_n;
                        (* Entry 'Default': '<S41>:7' *)
                        (* '<S41>:7:2' REQ_HV_ON = 0 *)
                        REQ_HV_ON := 0.0;
                        (* '<S41>:7:3' ContactorState = 1 *)
                        ContactorState := 1.0;
                    ELSE 
                        (* '<S41>:21:1' sf_internal_predicateOutput = after(2,sec) &&... *)
                        (* '<S41>:21:2' IMD_Active_BB1 == false &&... *)
                        (* '<S41>:21:3' IMD_Active_BB2 == true &&... *)
                        (* '<S41>:21:4' IMD_Active_BB3 == false &&... *)
                        (* '<S41>:21:5' MainHV_PlusMinus_Status == 0; *)
                        temporalCounter_i1(timerAction := 2, maxTime := 2000);

                        IF temporalCounter_i1.done THEN 

                            IF ((( NOT IMD_Active_BB1) AND IMD_Active_BB2) AND ( NOT IMD_Active_BB3)) AND ( NOT MainHV_PlusMinus_Status) THEN 
                                (* Transition: '<S41>:21' *)
                                temp3 := TRUE;
                            ELSE 
                                temp5 := TRUE;
                            END_IF;

                        ELSE 
                            temp5 := TRUE;
                        END_IF;

                    END_IF;

                ChiefMaster_IN_CONTACTOR_ON_o: 
                    (* During 'CONTACTOR_ON': '<S41>:20' *)
                    (* '<S41>:44:1' sf_internal_predicateOutput = (KL15_CM_disable == true || SDError_BB == true || System_SD == true) &&... *)
                    (* '<S41>:44:2' (MainHV_SD_OK == true || HV_REL_ON_BB2 == false); *)
                    tmp :=  NOT HV_REL_ON_BB2;

                    IF ((KL15_CM_disable OR SDError_BB) OR System_SD) AND (MainHV_SD_OK OR tmp) THEN 
                        (* Transition: '<S41>:44' *)
                        is_c5_ChiefMaster := ChiefMaster_IN_hold_i;
                        temporalCounter_i1(timerAction := 1, maxTime := 0);
                    ELSE 
                        (* '<S41>:51:1' sf_internal_predicateOutput = SDError_BB == true &&... *)
                        (* '<S41>:51:2' (HV_REL_ON_BB1 == true || HV_REL_ON_BB3 == true) &&... *)
                        (* '<S41>:51:3' (SafeToSD == true || HV_REL_ON_BB2 == false); *)
                        temp1 := HV_REL_ON_BB1 OR HV_REL_ON_BB3;

                        IF (SDError_BB AND temp1) AND (SafeToSD OR tmp) THEN 
                            (* Transition: '<S41>:51' *)
                            temp4 := TRUE;
                        ELSE 
                            (* '<S41>:66:1' sf_internal_predicateOutput = (HV_REL_ON_BB1 == true || HV_REL_ON_BB3 == true) &&... *)
                            (* '<S41>:66:2' REQ_HV_Open == true; *)

                            IF temp1 AND REQ_HV_Open THEN 
                                (* Transition: '<S41>:66' *)
                                temp4 := TRUE;
                            ELSE 
                                (* '<S41>:20:2' REQ_HV_ON = 1 *)
                                REQ_HV_ON := 1.0;
                                (* '<S41>:20:3' ContactorState = 3 *)
                                ContactorState := 3.0;
                            END_IF;

                        END_IF;

                    END_IF;

                b_ChiefMaster_IN_Default_n: 
                    (* During 'Default': '<S41>:7' *)
                    (* '<S41>:19:1' sf_internal_predicateOutput = IP_boChargeStop_Pressed == false &&... *)
                    (* '<S41>:19:2' KL15_CM_disable == false &&... *)
                    (* '<S41>:19:3' InsulationReadyOK == true &&... *)
                    (* '<S41>:19:4' SDError_BB == false &&... *)
                    (* '<S41>:19:5' System_SD == false; *)

                    IF (((( NOT IP_boChargeStop_Pressed) AND ( NOT KL15_CM_disable)) AND InsulationReadyOK) AND ( NOT SDError_BB)) AND ( NOT System_SD) THEN 
                        (* Transition: '<S41>:19' *)
                        is_c5_ChiefMaster := ChiefMaster_IN_CONTACTOR_OFF_p;
                        temporalCounter_i1(timerAction := 1, maxTime := 0);
                        temporalCounter_i2(timerAction := 1, maxTime := 0);
                        (* Entry 'CONTACTOR_OFF': '<S41>:18' *)
                        (* '<S41>:18:2' REQ_HV_ON = 0 *)
                        REQ_HV_ON := 0.0;
                        (* '<S41>:18:3' ContactorState = 2 *)
                        ContactorState := 2.0;
                    ELSE 
                        (* '<S41>:7:2' REQ_HV_ON = 0 *)
                        REQ_HV_ON := 0.0;
                        (* '<S41>:7:3' ContactorState = 1 *)
                        ContactorState := 1.0;
                    END_IF;

                ELSE
                    (* During 'hold': '<S41>:63' *)
                    (* '<S41>:64:1' sf_internal_predicateOutput = after(2,sec); *)
                    temporalCounter_i1(timerAction := 2, maxTime := 2000);

                    IF temporalCounter_i1.done THEN 
                        (* Transition: '<S41>:64' *)
                        is_c5_ChiefMaster := b_ChiefMaster_IN_Default_n;
                        (* Entry 'Default': '<S41>:7' *)
                        (* '<S41>:7:2' REQ_HV_ON = 0 *)
                        REQ_HV_ON := 0.0;
                        (* '<S41>:7:3' ContactorState = 1 *)
                        ContactorState := 1.0;
                    END_IF;

            END_CASE;


            IF temp5 THEN 
                (* '<S41>:28:1' sf_internal_predicateOutput = after(2,sec) &&... *)
                (* '<S41>:28:2' IMD_Active_BB2 == false &&... *)
                (* '<S41>:28:3' MainHV_PlusMinus_Status == 1 &&... *)
                (* '<S41>:28:4' (IMD_Active_BB1 == true || IMD_Active_BB3 ==true || IsolationMeasurementRequest == false) &&... *)
                (* '<S41>:28:5' SafeToCloseHV == true; *)
                temporalCounter_i2(timerAction := 2, maxTime := 2000);

                IF temporalCounter_i2.done THEN 

                    IF ((( NOT IMD_Active_BB2) AND MainHV_PlusMinus_Status) AND ((IMD_Active_BB1 OR IMD_Active_BB3) OR ( NOT IsolationMeasurementRequest))) AND SafeToCloseHV_f THEN 
                        (* Transition: '<S41>:28' *)
                        temp3 := TRUE;
                    ELSE 
                        temp2 := TRUE;
                    END_IF;

                ELSE 
                    temp2 := TRUE;
                END_IF;

            END_IF;


            IF temp4 THEN 
                is_c5_ChiefMaster := b_ChiefMaster_IN_Default_n;
                (* Entry 'Default': '<S41>:7' *)
                (* '<S41>:7:2' REQ_HV_ON = 0 *)
                REQ_HV_ON := 0.0;
                (* '<S41>:7:3' ContactorState = 1 *)
                ContactorState := 1.0;
            END_IF;


            IF temp3 THEN 
                is_c5_ChiefMaster := ChiefMaster_IN_CONTACTOR_ON_o;
                (* Entry 'CONTACTOR_ON': '<S41>:20' *)
                (* '<S41>:20:2' REQ_HV_ON = 1 *)
                REQ_HV_ON := 1.0;
                (* '<S41>:20:3' ContactorState = 3 *)
                ContactorState := 3.0;
            END_IF;


            IF temp2 THEN 
                (* '<S41>:18:2' REQ_HV_ON = 0 *)
                REQ_HV_ON := 0.0;
                (* '<S41>:18:3' ContactorState = 2 *)
                ContactorState := 2.0;
            END_IF;

        END_IF;

        (* End of Chart: '<S33>/Chart_REQ_HV_ON_Batt2 ' *)
END_CASE;

END_FUNCTION_BLOCK

// Device/Application/Chart_ContactorFB_State_Batt2
FUNCTION_BLOCK Chart_ContactorFB_State_Batt2
VAR_INPUT
	ssMethodType: SINT;
	HV_Minus_Sense_BB: BOOL;
	HV_Plus_Sense_BB: BOOL;
	REQ_HV_ON: LREAL;
END_VAR
VAR_OUTPUT
	Contactor_FB_State: LREAL;
END_VAR
VAR
	temporalCounter_i1: PLC_CODER_TIMER;
	is_c36_ChiefMaster: USINT;
	is_active_c36_ChiefMaster: USINT;
END_VAR



CASE ssMethodType OF
    SS_INITIALIZE: 
        temporalCounter_i1(timerAction := 1, maxTime := 0);
        is_active_c36_ChiefMaster := 0;
        is_c36_ChiefMaster := ChiefMaster_IN_NO_ACTIVE_CHILD_hs;
        Contactor_FB_State := 0.0;
    SS_OUTPUT: 
        (* Chart: '<S33>/Chart_ContactorFB_State_Batt2' *)
        (* Gateway: ChiefMaster/Flow Logic/Battery HVControl/REQ_HV_ON_Batt/Chart_ContactorFB_State_Batt2 *)
        (* During: ChiefMaster/Flow Logic/Battery HVControl/REQ_HV_ON_Batt/Chart_ContactorFB_State_Batt2 *)

        IF is_active_c36_ChiefMaster = 0 THEN 
            (* Entry: ChiefMaster/Flow Logic/Battery HVControl/REQ_HV_ON_Batt/Chart_ContactorFB_State_Batt2 *)
            is_active_c36_ChiefMaster := 1;
            (* Entry Internal: ChiefMaster/Flow Logic/Battery HVControl/REQ_HV_ON_Batt/Chart_ContactorFB_State_Batt2 *)
            (* Transition: '<S38>:2' *)
            is_c36_ChiefMaster := ChiefMaster_IN_default_h;
            (* Entry 'default': '<S38>:1' *)
            (* '<S38>:1:2' Contactor_FB_State = 0 *)
            Contactor_FB_State := 0.0;
        ELSE 

            CASE is_c36_ChiefMaster OF
                ChiefMaster_IN_Error_e: 
                    (* During 'Error': '<S38>:12' *)
                    (* '<S38>:51:1' sf_internal_predicateOutput = REQ_HV_ON == 1; *)

                    IF REQ_HV_ON = 1.0 THEN 
                        (* Transition: '<S38>:51' *)
                        is_c36_ChiefMaster := ChiefMaster_IN_default_h;
                        (* Entry 'default': '<S38>:1' *)
                        (* '<S38>:1:2' Contactor_FB_State = 0 *)
                        Contactor_FB_State := 0.0;
                    ELSE 
                        (* '<S38>:12:2' Contactor_FB_State = 3 *)
                        Contactor_FB_State := 3.0;
                    END_IF;

                ChiefMaster_IN_Open_p: 
                    (* During 'Open': '<S38>:46' *)
                    (* '<S38>:50:1' sf_internal_predicateOutput = REQ_HV_ON == 1; *)

                    IF REQ_HV_ON = 1.0 THEN 
                        (* Transition: '<S38>:50' *)
                        is_c36_ChiefMaster := ChiefMaster_IN_default_h;
                        (* Entry 'default': '<S38>:1' *)
                        (* '<S38>:1:2' Contactor_FB_State = 0 *)
                        Contactor_FB_State := 0.0;
                    ELSE 
                        (* '<S38>:46:2' Contactor_FB_State = 1 *)
                        Contactor_FB_State := 1.0;
                    END_IF;

                ChiefMaster_IN_default_h: 
                    (* During 'default': '<S38>:1' *)
                    (* '<S38>:5:1' sf_internal_predicateOutput = REQ_HV_ON == 0; *)

                    IF REQ_HV_ON = 0.0 THEN 
                        (* Transition: '<S38>:5' *)
                        is_c36_ChiefMaster := ChiefMaster_IN_hold_o;
                        temporalCounter_i1(timerAction := 1, maxTime := 0);
                        (* Entry 'hold': '<S38>:4' *)
                        (* '<S38>:4:2' Contactor_FB_State = 0 *)
                        Contactor_FB_State := 0.0;
                    ELSE 
                        (* '<S38>:1:2' Contactor_FB_State = 0 *)
                        Contactor_FB_State := 0.0;
                    END_IF;

                ELSE
                    (* During 'hold': '<S38>:4' *)
                    (* '<S38>:13:1' sf_internal_predicateOutput = after(5,sec); *)
                    temporalCounter_i1(timerAction := 2, maxTime := 5000);

                    IF temporalCounter_i1.done THEN 
                        (* Transition: '<S38>:13' *)
                        is_c36_ChiefMaster := ChiefMaster_IN_Error_e;
                        (* Entry 'Error': '<S38>:12' *)
                        (* '<S38>:12:2' Contactor_FB_State = 3 *)
                        Contactor_FB_State := 3.0;
                    ELSE 
                        (* '<S38>:47:1' sf_internal_predicateOutput = HV_Plus_Sense_BB == false &&... *)
                        (* '<S38>:47:2' HV_Minus_Sense_BB == false; *)

                        IF ( NOT HV_Plus_Sense_BB) AND ( NOT HV_Minus_Sense_BB) THEN 
                            (* Transition: '<S38>:47' *)
                            is_c36_ChiefMaster := ChiefMaster_IN_Open_p;
                            (* Entry 'Open': '<S38>:46' *)
                            (* '<S38>:46:2' Contactor_FB_State = 1 *)
                            Contactor_FB_State := 1.0;
                        ELSE 
                            (* '<S38>:4:2' Contactor_FB_State = 0 *)
                            Contactor_FB_State := 0.0;
                        END_IF;

                    END_IF;

            END_CASE;

        END_IF;

        (* End of Chart: '<S33>/Chart_ContactorFB_State_Batt2' *)
END_CASE;

END_FUNCTION_BLOCK

// Device/Application/Chart_REQ_HV_ON_Batt3
FUNCTION_BLOCK Chart_REQ_HV_ON_Batt3
VAR_INPUT
	ssMethodType: SINT;
	IP_boChargeStop_Pressed: BOOL;
	InsulationReadyOK: BOOL;
	SDError_BB: BOOL;
	IMD_Active_BB1: BOOL;
	IMD_Active_BB2: BOOL;
	IMD_Active_BB3: BOOL;
	Software_Reset_KL15_BB: LREAL;
	KL15_CM_disable: BOOL;
	SafeToCloseHV_n: BOOL;
	MainHV_SD_OK: BOOL;
	SafeToSD: BOOL;
	HV_REL_ON_BB1: BOOL;
	HV_REL_ON_BB2: BOOL;
	System_SD: BOOL;
	HV_REL_ON_BB3: BOOL;
	MainHV_PlusMinus_Status: BOOL;
	IsolationMeasurementRequest: BOOL;
	REQ_HV_Open: BOOL;
END_VAR
VAR_OUTPUT
	REQ_HV_ON: LREAL;
	ContactorState: LREAL;
END_VAR
VAR
	temporalCounter_i1: PLC_CODER_TIMER;
	temporalCounter_i2: PLC_CODER_TIMER;
	is_c6_ChiefMaster: USINT;
	is_active_c6_ChiefMaster: USINT;
	tmp: BOOL;
	temp1: BOOL;
	temp2: BOOL;
	temp3: BOOL;
	temp4: BOOL;
	temp5: BOOL;
END_VAR



